  LIN {X -15849.996,Y 231.529,Z 80.709,A 172.46345,B 0.00000,C -180.00000} ; retreat
  ; Step 2908, bar 3026
  LIN {X -15449.996,Y 231.529,Z 999.647,A 172.46345,B 0.00000,C -180.00000} ; outside
  LIN {X -15449.996,Y 231.529,Z 30.709,A 172.46345,B 0.00000,C -180.00000} ; preinsert
  LIN {X -15449.996,Y 231.529,Z -219.291,A 172.46345,B 0.00000,C -180.00000} ; insert
  LIN {X -15449.996,Y 231.529,Z -219.291,A 172.46345,B 0.00000,C -180.00000} ; release
  LIN {X -15449.996,Y 231.529,Z 80.709,A 172.46345,B 0.00000,C -180.00000} ; retreat
  ; Step 2909, bar 3059
  LIN {X 15449.996,Y 231.529,Z 999.648,A 7.53655,B 0.00000,C 180.00000} ; outside
  LIN {X 15449.996,Y 231.529,Z 30.709,A 7.53655,B 0.00000,C 180.00000} ; preinsert
  LIN {X 15449.996,Y 231.529,Z -219.291,A 7.53655,B 0.00000,C 180.00000} ; insert
  LIN {X 15449.996,Y 231.529,Z -219.291,A 7.53655,B 0.00000,C 180.00000} ; release
  LIN {X 15449.996,Y 231.529,Z 80.709,A 7.53655,B 0.00000,C 180.00000} ; retreat
  ; Step 2910, bar 3065
  LIN {X 15849.996,Y 231.529,Z 999.648,A 7.53655,B 0.00000,C 180.00000} ; outside
  LIN {X 15849.996,Y 231.529,Z 30.709,A 7.53655,B 0.00000,C 180.00000} ; preinsert
  LIN {X 15849.996,Y 231.529,Z -219.291,A 7.53655,B 0.00000,C 180.00000} ; insert
  LIN {X 15849.996,Y 231.529,Z -219.291,A 7.53655,B 0.00000,C 180.00000} ; release
  LIN {X 15849.996,Y 231.529,Z 80.709,A 7.53655,B 0.00000,C 180.00000} ; retreat
  ; Step 2911, bar 3071
  LIN {X 16249.996,Y 231.529,Z 999.648,A 7.53655,B 0.00000,C 180.00000} ; outside
  LIN {X 16249.996,Y 231.529,Z 30.709,A 7.53655,B 0.00000,C 180.00000} ; preinsert
  LIN {X 16249.996,Y 231.529,Z -219.291,A 7.53655,B 0.00000,C 180.00000} ; insert
  LIN {X 16249.996,Y 231.529,Z -219.291,A 7.53655,B 0.00000,C 180.00000} ; release
  LIN {X 16249.996,Y 231.529,Z 80.709,A 7.53655,B 0.00000,C 180.00000} ; retreat
  ; Step 2912, bar 2635
  LIN {X -11999.916,Y -18.207,Z 1090.744,A -87.44234,B 0.00000,C 180.00000} ; outside
  LIN {X -11999.916,Y -18.207,Z 121.634,A -87.44234,B 0.00000,C 180.00000} ; preinsert
  LIN {X -11999.916,Y -18.207,Z -128.366,A -87.44234,B 0.00000,C 180.00000} ; insert
  LIN {X -11999.916,Y -18.207,Z -128.366,A -87.44234,B 0.00000,C 180.00000} ; release
  LIN {X -11999.916,Y -18.207,Z 171.634,A -87.44234,B 0.00000,C 180.00000} ; retreat
  ; Step 2913, bar 2629
  LIN {X -11249.916,Y -18.207,Z 1090.744,A -87.44234,B 0.00000,C 180.00000} ; outside
  LIN {X -11249.916,Y -18.207,Z 121.634,A -87.44234,B 0.00000,C 180.00000} ; preinsert
  LIN {X -11249.916,Y -18.207,Z -128.366,A -87.44234,B 0.00000,C 180.00000} ; insert
  LIN {X -11249.916,Y -18.207,Z -128.366,A -87.44234,B 0.00000,C 180.00000} ; release
  LIN {X -11249.916,Y -18.207,Z 171.634,A -87.44234,B 0.00000,C 180.00000} ; retreat
  ; Step 2914, bar 2622
  LIN {X -10499.916,Y -18.207,Z 1090.744,A -87.44234,B 0.00000,C 180.00000} ; outside
  LIN {X -10499.916,Y -18.207,Z 121.634,A -87.44234,B 0.00000,C 180.00000} ; preinsert
  LIN {X -10499.916,Y -18.207,Z -128.366,A -87.44234,B 0.00000,C 180.00000} ; insert
  LIN {X -10499.916,Y -18.207,Z -128.366,A -87.44234,B 0.00000,C 180.00000} ; release
  LIN {X -10499.916,Y -18.207,Z 171.634,A -87.44234,B 0.00000,C 180.00000} ; retreat
  ; Step 2915, bar 2615
  LIN {X -9749.916,Y -18.207,Z 1090.744,A -87.44234,B 0.00000,C 180.00000} ; outside
  LIN {X -9749.916,Y -18.207,Z 121.634,A -87.44234,B 0.00000,C 180.00000} ; preinsert
  LIN {X -9749.916,Y -18.207,Z -128.366,A -87.44234,B 0.00000,C 180.00000} ; insert
  LIN {X -9749.916,Y -18.207,Z -128.366,A -87.44234,B 0.00000,C 180.00000} ; release
  LIN {X -9749.916,Y -18.207,Z 171.634,A -87.44234,B 0.00000,C 180.00000} ; retreat
  ; Step 2916, bar 2608
  LIN {X -8999.916,Y -18.207,Z 1090.744,A -87.44234,B 0.00000,C 180.00000} ; outside
  LIN {X -8999.916,Y -18.207,Z 121.634,A -87.44234,B 0.00000,C 180.00000} ; preinsert
  LIN {X -8999.916,Y -18.207,Z -128.366,A -87.44234,B 0.00000,C 180.00000} ; insert
  LIN {X -8999.916,Y -18.207,Z -128.366,A -87.44234,B 0.00000,C 180.00000} ; release
  LIN {X -8999.916,Y -18.207,Z 171.634,A -87.44234,B 0.00000,C 180.00000} ; retreat
  ; Step 2917, bar 2601
  LIN {X -8249.916,Y -18.207,Z 1090.744,A -87.44234,B 0.00000,C 180.00000} ; outside
  LIN {X -8249.916,Y -18.207,Z 121.634,A -87.44234,B 0.00000,C 180.00000} ; preinsert
  LIN {X -8249.916,Y -18.207,Z -128.366,A -87.44234,B 0.00000,C 180.00000} ; insert
  LIN {X -8249.916,Y -18.207,Z -128.366,A -87.44234,B 0.00000,C 180.00000} ; release
  LIN {X -8249.916,Y -18.207,Z 171.634,A -87.44234,B 0.00000,C 180.00000} ; retreat
  ; Step 2918, bar 2594
  LIN {X -7499.916,Y -18.207,Z 1090.744,A -87.44234,B 0.00000,C 180.00000} ; outside
  LIN {X -7499.916,Y -18.207,Z 121.634,A -87.44234,B 0.00000,C 180.00000} ; preinsert
  LIN {X -7499.916,Y -18.207,Z -128.366,A -87.44234,B 0.00000,C 180.00000} ; insert
  LIN {X -7499.916,Y -18.207,Z -128.366,A -87.44234,B 0.00000,C 180.00000} ; release
  LIN {X -7499.916,Y -18.207,Z 171.634,A -87.44234,B 0.00000,C 180.00000} ; retreat
  ; Step 2919, bar 2587
  LIN {X -6749.916,Y -18.207,Z 1090.744,A -87.44234,B 0.00000,C 180.00000} ; outside
  LIN {X -6749.916,Y -18.207,Z 121.634,A -87.44234,B 0.00000,C 180.00000} ; preinsert
  LIN {X -6749.916,Y -18.207,Z -128.366,A -87.44234,B 0.00000,C 180.00000} ; insert
  LIN {X -6749.916,Y -18.207,Z -128.366,A -87.44234,B 0.00000,C 180.00000} ; release
  LIN {X -6749.916,Y -18.207,Z 171.634,A -87.44234,B 0.00000,C 180.00000} ; retreat
  ; Step 2920, bar 2580
  LIN {X -5999.916,Y -18.207,Z 1090.744,A -87.44234,B 0.00000,C 180.00000} ; outside
  LIN {X -5999.916,Y -18.207,Z 121.634,A -87.44234,B 0.00000,C 180.00000} ; preinsert
  LIN {X -5999.916,Y -18.207,Z -128.366,A -87.44234,B 0.00000,C 180.00000} ; insert
  LIN {X -5999.916,Y -18.207,Z -128.366,A -87.44234,B 0.00000,C 180.00000} ; release
  LIN {X -5999.916,Y -18.207,Z 171.634,A -87.44234,B 0.00000,C 180.00000} ; retreat
  ; Step 2921, bar 2573
  LIN {X -5249.916,Y -18.207,Z 1090.744,A -87.44234,B 0.00000,C 180.00000} ; outside
  LIN {X -5249.916,Y -18.207,Z 121.634,A -87.44234,B 0.00000,C 180.00000} ; preinsert
  LIN {X -5249.916,Y -18.207,Z -128.366,A -87.44234,B 0.00000,C 180.00000} ; insert
  LIN {X -5249.916,Y -18.207,Z -128.366,A -87.44234,B 0.00000,C 180.00000} ; release
  LIN {X -5249.916,Y -18.207,Z 171.634,A -87.44234,B 0.00000,C 180.00000} ; retreat
  ; Step 2922, bar 2566
  LIN {X -4499.916,Y -18.207,Z 1090.744,A -87.44234,B 0.00000,C 180.00000} ; outside
  LIN {X -4499.916,Y -18.207,Z 121.634,A -87.44234,B 0.00000,C 180.00000} ; preinsert
  LIN {X -4499.916,Y -18.207,Z -128.366,A -87.44234,B 0.00000,C 180.00000} ; insert
  LIN {X -4499.916,Y -18.207,Z -128.366,A -87.44234,B 0.00000,C 180.00000} ; release
  LIN {X -4499.916,Y -18.207,Z 171.634,A -87.44234,B 0.00000,C 180.00000} ; retreat
  ; Step 2923, bar 2559
  LIN {X -3749.916,Y -18.207,Z 1090.744,A -87.44234,B 0.00000,C 180.00000} ; outside
  LIN {X -3749.916,Y -18.207,Z 121.634,A -87.44234,B 0.00000,C 180.00000} ; preinsert
  LIN {X -3749.916,Y -18.207,Z -128.366,A -87.44234,B 0.00000,C 180.00000} ; insert
  LIN {X -3749.916,Y -18.207,Z -128.366,A -87.44234,B 0.00000,C 180.00000} ; release
  LIN {X -3749.916,Y -18.207,Z 171.634,A -87.44234,B 0.00000,C 180.00000} ; retreat
  ; Step 2924, bar 2552
  LIN {X -2999.916,Y -18.207,Z 1090.744,A -87.44234,B 0.00000,C 180.00000} ; outside
  LIN {X -2999.916,Y -18.207,Z 121.634,A -87.44234,B 0.00000,C 180.00000} ; preinsert
  LIN {X -2999.916,Y -18.207,Z -128.366,A -87.44234,B 0.00000,C 180.00000} ; insert
  LIN {X -2999.916,Y -18.207,Z -128.366,A -87.44234,B 0.00000,C 180.00000} ; release
  LIN {X -2999.916,Y -18.207,Z 171.634,A -87.44234,B 0.00000,C 180.00000} ; retreat
  ; Step 2925, bar 2545
  LIN {X -2249.916,Y -18.207,Z 1090.744,A -87.44234,B 0.00000,C 180.00000} ; outside
  LIN {X -2249.916,Y -18.207,Z 121.634,A -87.44234,B 0.00000,C 180.00000} ; preinsert
  LIN {X -2249.916,Y -18.207,Z -128.366,A -87.44234,B 0.00000,C 180.00000} ; insert
  LIN {X -2249.916,Y -18.207,Z -128.366,A -87.44234,B 0.00000,C 180.00000} ; release
  LIN {X -2249.916,Y -18.207,Z 171.634,A -87.44234,B 0.00000,C 180.00000} ; retreat
  ; Step 2926, bar 2538
  LIN {X -1499.916,Y -18.207,Z 1090.744,A -87.44234,B 0.00000,C 180.00000} ; outside
  LIN {X -1499.916,Y -18.207,Z 121.634,A -87.44234,B 0.00000,C 180.00000} ; preinsert
  LIN {X -1499.916,Y -18.207,Z -128.366,A -87.44234,B 0.00000,C 180.00000} ; insert
  LIN {X -1499.916,Y -18.207,Z -128.366,A -87.44234,B 0.00000,C 180.00000} ; release
  LIN {X -1499.916,Y -18.207,Z 171.634,A -87.44234,B 0.00000,C 180.00000} ; retreat
  ; Step 2927, bar 1972
  LIN {X 0.084,Y -18.207,Z 1090.744,A -87.44234,B 0.00000,C -180.00000} ; outside
  LIN {X 0.084,Y -18.207,Z 121.634,A -87.44234,B 0.00000,C -180.00000} ; preinsert
  LIN {X 0.084,Y -18.207,Z -128.366,A -87.44234,B 0.00000,C -180.00000} ; insert
  LIN {X 0.084,Y -18.207,Z -128.366,A -87.44234,B 0.00000,C -180.00000} ; release
  LIN {X 0.084,Y -18.207,Z 171.634,A -87.44234,B 0.00000,C -180.00000} ; retreat
  ; Step 2928, bar 2691
  LIN {X 1499.916,Y -18.207,Z 1090.744,A -92.55766,B 0.00000,C -180.00000} ; outside
  LIN {X 1499.916,Y -18.207,Z 121.634,A -92.55766,B 0.00000,C -180.00000} ; preinsert
  LIN {X 1499.916,Y -18.207,Z -128.366,A -92.55766,B 0.00000,C -180.00000} ; insert
  LIN {X 1499.916,Y -18.207,Z -128.366,A -92.55766,B 0.00000,C -180.00000} ; release
  LIN {X 1499.916,Y -18.207,Z 171.634,A -92.55766,B 0.00000,C -180.00000} ; retreat
  ; Step 2929, bar 2695
  LIN {X 2249.916,Y -18.207,Z 1090.744,A -92.55766,B 0.00000,C -180.00000} ; outside
  LIN {X 2249.916,Y -18.207,Z 121.634,A -92.55766,B 0.00000,C -180.00000} ; preinsert
  LIN {X 2249.916,Y -18.207,Z -128.366,A -92.55766,B 0.00000,C -180.00000} ; insert
  LIN {X 2249.916,Y -18.207,Z -128.366,A -92.55766,B 0.00000,C -180.00000} ; release
  LIN {X 2249.916,Y -18.207,Z 171.634,A -92.55766,B 0.00000,C -180.00000} ; retreat
  ; Step 2930, bar 2699
  LIN {X 2999.916,Y -18.207,Z 1090.744,A -92.55766,B 0.00000,C -180.00000} ; outside
  LIN {X 2999.916,Y -18.207,Z 121.634,A -92.55766,B 0.00000,C -180.00000} ; preinsert
  LIN {X 2999.916,Y -18.207,Z -128.366,A -92.55766,B 0.00000,C -180.00000} ; insert
  LIN {X 2999.916,Y -18.207,Z -128.366,A -92.55766,B 0.00000,C -180.00000} ; release
  LIN {X 2999.916,Y -18.207,Z 171.634,A -92.55766,B 0.00000,C -180.00000} ; retreat
  ; Step 2931, bar 2703
  LIN {X 3749.916,Y -18.207,Z 1090.744,A -92.55766,B 0.00000,C -180.00000} ; outside
  LIN {X 3749.916,Y -18.207,Z 121.634,A -92.55766,B 0.00000,C -180.00000} ; preinsert
  LIN {X 3749.916,Y -18.207,Z -128.366,A -92.55766,B 0.00000,C -180.00000} ; insert
  LIN {X 3749.916,Y -18.207,Z -128.366,A -92.55766,B 0.00000,C -180.00000} ; release
  LIN {X 3749.916,Y -18.207,Z 171.634,A -92.55766,B 0.00000,C -180.00000} ; retreat
  ; Step 2932, bar 2707
  LIN {X 4499.916,Y -18.207,Z 1090.744,A -92.55766,B 0.00000,C -180.00000} ; outside
  LIN {X 4499.916,Y -18.207,Z 121.634,A -92.55766,B 0.00000,C -180.00000} ; preinsert
  LIN {X 4499.916,Y -18.207,Z -128.366,A -92.55766,B 0.00000,C -180.00000} ; insert
  LIN {X 4499.916,Y -18.207,Z -128.366,A -92.55766,B 0.00000,C -180.00000} ; release
  LIN {X 4499.916,Y -18.207,Z 171.634,A -92.55766,B 0.00000,C -180.00000} ; retreat
  ; Step 2933, bar 2711
  LIN {X 5249.916,Y -18.207,Z 1090.744,A -92.55766,B 0.00000,C -180.00000} ; outside
  LIN {X 5249.916,Y -18.207,Z 121.634,A -92.55766,B 0.00000,C -180.00000} ; preinsert
  LIN {X 5249.916,Y -18.207,Z -128.366,A -92.55766,B 0.00000,C -180.00000} ; insert
  LIN {X 5249.916,Y -18.207,Z -128.366,A -92.55766,B 0.00000,C -180.00000} ; release
  LIN {X 5249.916,Y -18.207,Z 171.634,A -92.55766,B 0.00000,C -180.00000} ; retreat
  ; Step 2934, bar 2715
  LIN {X 5999.916,Y -18.207,Z 1090.744,A -92.55766,B 0.00000,C -180.00000} ; outside
  LIN {X 5999.916,Y -18.207,Z 121.634,A -92.55766,B 0.00000,C -180.00000} ; preinsert
  LIN {X 5999.916,Y -18.207,Z -128.366,A -92.55766,B 0.00000,C -180.00000} ; insert
  LIN {X 5999.916,Y -18.207,Z -128.366,A -92.55766,B 0.00000,C -180.00000} ; release
  LIN {X 5999.916,Y -18.207,Z 171.634,A -92.55766,B 0.00000,C -180.00000} ; retreat
  ; Step 2935, bar 2719
  LIN {X 6749.916,Y -18.207,Z 1090.744,A -92.55766,B 0.00000,C -180.00000} ; outside
  LIN {X 6749.916,Y -18.207,Z 121.634,A -92.55766,B 0.00000,C -180.00000} ; preinsert
  LIN {X 6749.916,Y -18.207,Z -128.366,A -92.55766,B 0.00000,C -180.00000} ; insert
  LIN {X 6749.916,Y -18.207,Z -128.366,A -92.55766,B 0.00000,C -180.00000} ; release
  LIN {X 6749.916,Y -18.207,Z 171.634,A -92.55766,B 0.00000,C -180.00000} ; retreat
  ; Step 2936, bar 2723
  LIN {X 7499.916,Y -18.207,Z 1090.744,A -92.55766,B 0.00000,C -180.00000} ; outside
  LIN {X 7499.916,Y -18.207,Z 121.634,A -92.55766,B 0.00000,C -180.00000} ; preinsert
  LIN {X 7499.916,Y -18.207,Z -128.366,A -92.55766,B 0.00000,C -180.00000} ; insert
  LIN {X 7499.916,Y -18.207,Z -128.366,A -92.55766,B 0.00000,C -180.00000} ; release
  LIN {X 7499.916,Y -18.207,Z 171.634,A -92.55766,B 0.00000,C -180.00000} ; retreat
  ; Step 2937, bar 2727
  LIN {X 8249.916,Y -18.207,Z 1090.744,A -92.55766,B 0.00000,C -180.00000} ; outside
  LIN {X 8249.916,Y -18.207,Z 121.634,A -92.55766,B 0.00000,C -180.00000} ; preinsert
  LIN {X 8249.916,Y -18.207,Z -128.366,A -92.55766,B 0.00000,C -180.00000} ; insert
  LIN {X 8249.916,Y -18.207,Z -128.366,A -92.55766,B 0.00000,C -180.00000} ; release
  LIN {X 8249.916,Y -18.207,Z 171.634,A -92.55766,B 0.00000,C -180.00000} ; retreat
  ; Step 2938, bar 2731
  LIN {X 8999.916,Y -18.207,Z 1090.744,A -92.55766,B 0.00000,C -180.00000} ; outside
  LIN {X 8999.916,Y -18.207,Z 121.634,A -92.55766,B 0.00000,C -180.00000} ; preinsert
  LIN {X 8999.916,Y -18.207,Z -128.366,A -92.55766,B 0.00000,C -180.00000} ; insert
  LIN {X 8999.916,Y -18.207,Z -128.366,A -92.55766,B 0.00000,C -180.00000} ; release
  LIN {X 8999.916,Y -18.207,Z 171.634,A -92.55766,B 0.00000,C -180.00000} ; retreat
  ; Step 2939, bar 2735
  LIN {X 9749.916,Y -18.207,Z 1090.744,A -92.55766,B 0.00000,C -180.00000} ; outside
  LIN {X 9749.916,Y -18.207,Z 121.634,A -92.55766,B 0.00000,C -180.00000} ; preinsert
  LIN {X 9749.916,Y -18.207,Z -128.366,A -92.55766,B 0.00000,C -180.00000} ; insert
  LIN {X 9749.916,Y -18.207,Z -128.366,A -92.55766,B 0.00000,C -180.00000} ; release
  LIN {X 9749.916,Y -18.207,Z 171.634,A -92.55766,B 0.00000,C -180.00000} ; retreat
  ; Step 2940, bar 2739
  LIN {X 10499.916,Y -18.207,Z 1090.744,A -92.55766,B 0.00000,C -180.00000} ; outside
  LIN {X 10499.916,Y -18.207,Z 121.634,A -92.55766,B 0.00000,C -180.00000} ; preinsert
  LIN {X 10499.916,Y -18.207,Z -128.366,A -92.55766,B 0.00000,C -180.00000} ; insert
  LIN {X 10499.916,Y -18.207,Z -128.366,A -92.55766,B 0.00000,C -180.00000} ; release
  LIN {X 10499.916,Y -18.207,Z 171.634,A -92.55766,B 0.00000,C -180.00000} ; retreat
  ; Step 2941, bar 2743
  LIN {X 11249.916,Y -18.207,Z 1090.744,A -92.55766,B 0.00000,C -180.00000} ; outside
  LIN {X 11249.916,Y -18.207,Z 121.634,A -92.55766,B 0.00000,C -180.00000} ; preinsert
  LIN {X 11249.916,Y -18.207,Z -128.366,A -92.55766,B 0.00000,C -180.00000} ; insert
  LIN {X 11249.916,Y -18.207,Z -128.366,A -92.55766,B 0.00000,C -180.00000} ; release
  LIN {X 11249.916,Y -18.207,Z 171.634,A -92.55766,B 0.00000,C -180.00000} ; retreat
  ; Step 2942, bar 2747
  LIN {X 11999.916,Y -18.207,Z 1090.744,A -92.55766,B 0.00000,C -180.00000} ; outside
  LIN {X 11999.916,Y -18.207,Z 121.634,A -92.55766,B 0.00000,C -180.00000} ; preinsert
  LIN {X 11999.916,Y -18.207,Z -128.366,A -92.55766,B 0.00000,C -180.00000} ; insert
  LIN {X 11999.916,Y -18.207,Z -128.366,A -92.55766,B 0.00000,C -180.00000} ; release
  LIN {X 11999.916,Y -18.207,Z 171.634,A -92.55766,B 0.00000,C -180.00000} ; retreat
  ; Step 2943, bar 2687
  LIN {X 749.916,Y -18.207,Z 1090.744,A -92.55766,B 0.00000,C -180.00000} ; outside
  LIN {X 749.916,Y -18.207,Z 121.634,A -92.55766,B 0.00000,C -180.00000} ; preinsert
  LIN {X 749.916,Y -18.207,Z -128.366,A -92.55766,B 0.00000,C -180.00000} ; insert
  LIN {X 749.916,Y -18.207,Z -128.366,A -92.55766,B 0.00000,C -180.00000} ; release
  LIN {X 749.916,Y -18.207,Z 171.634,A -92.55766,B 0.00000,C -180.00000} ; retreat
  ; Step 2944, bar 2531
  LIN {X -749.916,Y -18.207,Z 1090.744,A -87.44234,B 0.00000,C 180.00000} ; outside
  LIN {X -749.916,Y -18.207,Z 121.634,A -87.44234,B 0.00000,C 180.00000} ; preinsert
  LIN {X -749.916,Y -18.207,Z -128.366,A -87.44234,B 0.00000,C 180.00000} ; insert
  LIN {X -749.916,Y -18.207,Z -128.366,A -87.44234,B 0.00000,C 180.00000} ; release
  LIN {X -749.916,Y -18.207,Z 171.634,A -87.44234,B 0.00000,C 180.00000} ; retreat
  ; Step 2945, bar 3056
  LIN {X 15249.996,Y -18.471,Z 1010.647,A 7.53655,B 0.00000,C 180.00000} ; outside
  LIN {X 15249.996,Y -18.471,Z 36.610,A 7.53655,B 0.00000,C 180.00000} ; preinsert
  LIN {X 15249.996,Y -18.471,Z -213.390,A 7.53655,B 0.00000,C 180.00000} ; insert
  LIN {X 15249.996,Y -18.471,Z -213.390,A 7.53655,B 0.00000,C 180.00000} ; release
  LIN {X 15249.996,Y -18.471,Z 86.610,A 7.53655,B 0.00000,C 180.00000} ; retreat
  ; Step 2946, bar 3062
  LIN {X 15649.996,Y -18.471,Z 1010.647,A 7.53655,B 0.00000,C 180.00000} ; outside
  LIN {X 15649.996,Y -18.471,Z 36.610,A 7.53655,B 0.00000,C 180.00000} ; preinsert
  LIN {X 15649.996,Y -18.471,Z -213.390,A 7.53655,B 0.00000,C 180.00000} ; insert
  LIN {X 15649.996,Y -18.471,Z -213.390,A 7.53655,B 0.00000,C 180.00000} ; release
  LIN {X 15649.996,Y -18.471,Z 86.610,A 7.53655,B 0.00000,C 180.00000} ; retreat
  ; Step 2947, bar 3068
  LIN {X 16049.996,Y -18.471,Z 1010.647,A 7.53655,B 0.00000,C 180.00000} ; outside
  LIN {X 16049.996,Y -18.471,Z 36.610,A 7.53655,B 0.00000,C 180.00000} ; preinsert
  LIN {X 16049.996,Y -18.471,Z -213.390,A 7.53655,B 0.00000,C 180.00000} ; insert
  LIN {X 16049.996,Y -18.471,Z -213.390,A 7.53655,B 0.00000,C 180.00000} ; release
  LIN {X 16049.996,Y -18.471,Z 86.610,A 7.53655,B 0.00000,C 180.00000} ; retreat
  ; Step 2948, bar 3035
  LIN {X -16049.996,Y -18.471,Z 1010.647,A 172.46345,B 0.00000,C 180.00000} ; outside
  LIN {X -16049.996,Y -18.471,Z 36.610,A 172.46345,B 0.00000,C 180.00000} ; preinsert
  LIN {X -16049.996,Y -18.471,Z -213.390,A 172.46345,B 0.00000,C 180.00000} ; insert
  LIN {X -16049.996,Y -18.471,Z -213.390,A 172.46345,B 0.00000,C 180.00000} ; release
  LIN {X -16049.996,Y -18.471,Z 86.610,A 172.46345,B 0.00000,C 180.00000} ; retreat
  ; Step 2949, bar 3029
  LIN {X -15649.996,Y -18.471,Z 1010.647,A 172.46345,B 0.00000,C 180.00000} ; outside
  LIN {X -15649.996,Y -18.471,Z 36.610,A 172.46345,B 0.00000,C 180.00000} ; preinsert
  LIN {X -15649.996,Y -18.471,Z -213.390,A 172.46345,B 0.00000,C 180.00000} ; insert
  LIN {X -15649.996,Y -18.471,Z -213.390,A 172.46345,B 0.00000,C 180.00000} ; release
  LIN {X -15649.996,Y -18.471,Z 86.610,A 172.46345,B 0.00000,C 180.00000} ; retreat
  ; Step 2950, bar 3023
  LIN {X -15249.996,Y -18.471,Z 1010.647,A 172.46345,B 0.00000,C 180.00000} ; outside
  LIN {X -15249.996,Y -18.471,Z 36.610,A 172.46345,B 0.00000,C 180.00000} ; preinsert
  LIN {X -15249.996,Y -18.471,Z -213.390,A 172.46345,B 0.00000,C 180.00000} ; insert
  LIN {X -15249.996,Y -18.471,Z -213.390,A 172.46345,B 0.00000,C 180.00000} ; release
  LIN {X -15249.996,Y -18.471,Z 86.610,A 172.46345,B 0.00000,C 180.00000} ; retreat
  ; Step 2951, bar 1530
  LIN {X 1986.216,Y 1384.682,Z 869.354,A -90.02766,B 0.00000,C -180.00000} ; outside
  LIN {X 1986.216,Y 1384.682,Z -118.655,A -90.02766,B 0.00000,C -180.00000} ; preinsert
  LIN {X 1986.216,Y 1384.682,Z -368.655,A -90.02766,B 0.00000,C -180.00000} ; insert
  LIN {X 1986.216,Y 1384.682,Z -368.655,A -90.02766,B 0.00000,C -180.00000} ; release
  LIN {X 1986.216,Y 1384.682,Z -68.655,A -90.02766,B 0.00000,C -180.00000} ; retreat
  ; Step 2952, bar 1532
  LIN {X 5986.216,Y 1384.682,Z 869.354,A -90.02766,B 0.00000,C 180.00000} ; outside
  LIN {X 5986.216,Y 1384.682,Z -118.655,A -90.02766,B 0.00000,C 180.00000} ; preinsert
  LIN {X 5986.216,Y 1384.682,Z -368.655,A -90.02766,B 0.00000,C 180.00000} ; insert
  LIN {X 5986.216,Y 1384.682,Z -368.655,A -90.02766,B 0.00000,C 180.00000} ; release
  LIN {X 5986.216,Y 1384.682,Z -68.655,A -90.02766,B 0.00000,C 180.00000} ; retreat
  ; Step 2953, bar 1534
  LIN {X 9986.216,Y 1384.682,Z 869.354,A -90.02766,B 0.00000,C -180.00000} ; outside
  LIN {X 9986.216,Y 1384.682,Z -118.655,A -90.02766,B 0.00000,C -180.00000} ; preinsert
  LIN {X 9986.216,Y 1384.682,Z -368.655,A -90.02766,B 0.00000,C -180.00000} ; insert
  LIN {X 9986.216,Y 1384.682,Z -368.655,A -90.02766,B 0.00000,C -180.00000} ; release
  LIN {X 9986.216,Y 1384.682,Z -68.655,A -90.02766,B 0.00000,C -180.00000} ; retreat
  ; Step 2954, bar 1536
  LIN {X 13936.216,Y 1384.682,Z 869.354,A -90.02766,B 0.00000,C -180.00000} ; outside
  LIN {X 13936.216,Y 1384.682,Z -118.655,A -90.02766,B 0.00000,C -180.00000} ; preinsert
  LIN {X 13936.216,Y 1384.682,Z -368.655,A -90.02766,B 0.00000,C -180.00000} ; insert
  LIN {X 13936.216,Y 1384.682,Z -368.655,A -90.02766,B 0.00000,C -180.00000} ; release
  LIN {X 13936.216,Y 1384.682,Z -68.655,A -90.02766,B 0.00000,C -180.00000} ; retreat
  ; Step 2955, bar 1538
  LIN {X 14036.216,Y 1384.682,Z 869.354,A -90.02766,B 0.00000,C -180.00000} ; outside
  LIN {X 14036.216,Y 1384.682,Z -118.655,A -90.02766,B 0.00000,C -180.00000} ; preinsert
  LIN {X 14036.216,Y 1384.682,Z -368.655,A -90.02766,B 0.00000,C -180.00000} ; insert
  LIN {X 14036.216,Y 1384.682,Z -368.655,A -90.02766,B 0.00000,C -180.00000} ; release
  LIN {X 14036.216,Y 1384.682,Z -68.655,A -90.02766,B 0.00000,C -180.00000} ; retreat
  ; Step 2956, bar 1549
  LIN {X -1986.216,Y -1384.682,Z 869.354,A 89.97234,B 0.00000,C 180.00000} ; outside
  LIN {X -1986.216,Y -1384.682,Z -118.655,A 89.97234,B 0.00000,C 180.00000} ; preinsert
  LIN {X -1986.216,Y -1384.682,Z -368.655,A 89.97234,B 0.00000,C 180.00000} ; insert
  LIN {X -1986.216,Y -1384.682,Z -368.655,A 89.97234,B 0.00000,C 180.00000} ; release
  LIN {X -1986.216,Y -1384.682,Z -68.655,A 89.97234,B 0.00000,C 180.00000} ; retreat
  ; Step 2957, bar 1551
  LIN {X -5986.216,Y -1384.682,Z 869.354,A 89.97234,B 0.00000,C 180.00000} ; outside
  LIN {X -5986.216,Y -1384.682,Z -118.655,A 89.97234,B 0.00000,C 180.00000} ; preinsert
  LIN {X -5986.216,Y -1384.682,Z -368.655,A 89.97234,B 0.00000,C 180.00000} ; insert
  LIN {X -5986.216,Y -1384.682,Z -368.655,A 89.97234,B 0.00000,C 180.00000} ; release
  LIN {X -5986.216,Y -1384.682,Z -68.655,A 89.97234,B 0.00000,C 180.00000} ; retreat
  ; Step 2958, bar 1553
  LIN {X -9986.216,Y -1384.682,Z 869.354,A 89.97234,B 0.00000,C -180.00000} ; outside
  LIN {X -9986.216,Y -1384.682,Z -118.655,A 89.97234,B 0.00000,C -180.00000} ; preinsert
  LIN {X -9986.216,Y -1384.682,Z -368.655,A 89.97234,B 0.00000,C -180.00000} ; insert
  LIN {X -9986.216,Y -1384.682,Z -368.655,A 89.97234,B 0.00000,C -180.00000} ; release
  LIN {X -9986.216,Y -1384.682,Z -68.655,A 89.97234,B 0.00000,C -180.00000} ; retreat
  ; Step 2959, bar 1555
  LIN {X -13936.216,Y -1384.682,Z 869.354,A 89.97234,B 0.00000,C -180.00000} ; outside
  LIN {X -13936.216,Y -1384.682,Z -118.655,A 89.97234,B 0.00000,C -180.00000} ; preinsert
  LIN {X -13936.216,Y -1384.682,Z -368.655,A 89.97234,B 0.00000,C -180.00000} ; insert
  LIN {X -13936.216,Y -1384.682,Z -368.655,A 89.97234,B 0.00000,C -180.00000} ; release
  LIN {X -13936.216,Y -1384.682,Z -68.655,A 89.97234,B 0.00000,C -180.00000} ; retreat
  ; Step 2960, bar 1557
  LIN {X -14036.216,Y -1384.682,Z 869.354,A 89.97234,B 0.00000,C -180.00000} ; outside
  LIN {X -14036.216,Y -1384.682,Z -118.655,A 89.97234,B 0.00000,C -180.00000} ; preinsert
  LIN {X -14036.216,Y -1384.682,Z -368.655,A 89.97234,B 0.00000,C -180.00000} ; insert
  LIN {X -14036.216,Y -1384.682,Z -368.655,A 89.97234,B 0.00000,C -180.00000} ; release
  LIN {X -14036.216,Y -1384.682,Z -68.655,A 89.97234,B 0.00000,C -180.00000} ; retreat
  ; Step 2961, bar 1529
  LIN {X 1986.216,Y -1384.663,Z 869.359,A 90.02766,B 0.00000,C 180.00000} ; outside
  LIN {X 1986.216,Y -1384.663,Z -118.650,A 90.02766,B 0.00000,C 180.00000} ; preinsert
  LIN {X 1986.216,Y -1384.663,Z -368.650,A 90.02766,B 0.00000,C 180.00000} ; insert
  LIN {X 1986.216,Y -1384.663,Z -368.650,A 90.02766,B 0.00000,C 180.00000} ; release
  LIN {X 1986.216,Y -1384.663,Z -68.650,A 90.02766,B 0.00000,C 180.00000} ; retreat
  ; Step 2962, bar 1531
  LIN {X 5986.216,Y -1384.663,Z 869.359,A 90.02766,B 0.00000,C 180.00000} ; outside
  LIN {X 5986.216,Y -1384.663,Z -118.650,A 90.02766,B 0.00000,C 180.00000} ; preinsert
  LIN {X 5986.216,Y -1384.663,Z -368.650,A 90.02766,B 0.00000,C 180.00000} ; insert
  LIN {X 5986.216,Y -1384.663,Z -368.650,A 90.02766,B 0.00000,C 180.00000} ; release
  LIN {X 5986.216,Y -1384.663,Z -68.650,A 90.02766,B 0.00000,C 180.00000} ; retreat
  ; Step 2963, bar 1533
  LIN {X 9986.216,Y -1384.663,Z 869.359,A 90.02766,B 0.00000,C -180.00000} ; outside
  LIN {X 9986.216,Y -1384.663,Z -118.650,A 90.02766,B 0.00000,C -180.00000} ; preinsert
  LIN {X 9986.216,Y -1384.663,Z -368.650,A 90.02766,B 0.00000,C -180.00000} ; insert
  LIN {X 9986.216,Y -1384.663,Z -368.650,A 90.02766,B 0.00000,C -180.00000} ; release
  LIN {X 9986.216,Y -1384.663,Z -68.650,A 90.02766,B 0.00000,C -180.00000} ; retreat
  ; Step 2964, bar 1535
  LIN {X 13936.216,Y -1384.663,Z 869.359,A 90.02766,B 0.00000,C -180.00000} ; outside
  LIN {X 13936.216,Y -1384.663,Z -118.650,A 90.02766,B 0.00000,C -180.00000} ; preinsert
  LIN {X 13936.216,Y -1384.663,Z -368.650,A 90.02766,B 0.00000,C -180.00000} ; insert
  LIN {X 13936.216,Y -1384.663,Z -368.650,A 90.02766,B 0.00000,C -180.00000} ; release
  LIN {X 13936.216,Y -1384.663,Z -68.650,A 90.02766,B 0.00000,C -180.00000} ; retreat
  ; Step 2965, bar 1537
  LIN {X 14036.216,Y -1384.663,Z 869.359,A 90.02766,B 0.00000,C -180.00000} ; outside
  LIN {X 14036.216,Y -1384.663,Z -118.650,A 90.02766,B 0.00000,C -180.00000} ; preinsert
  LIN {X 14036.216,Y -1384.663,Z -368.650,A 90.02766,B 0.00000,C -180.00000} ; insert
  LIN {X 14036.216,Y -1384.663,Z -368.650,A 90.02766,B 0.00000,C -180.00000} ; release
  LIN {X 14036.216,Y -1384.663,Z -68.650,A 90.02766,B 0.00000,C -180.00000} ; retreat
  ; Step 2966, bar 1550
  LIN {X -1986.216,Y 1384.663,Z 869.359,A -89.97234,B 0.00000,C 180.00000} ; outside
  LIN {X -1986.216,Y 1384.663,Z -118.650,A -89.97234,B 0.00000,C 180.00000} ; preinsert
  LIN {X -1986.216,Y 1384.663,Z -368.650,A -89.97234,B 0.00000,C 180.00000} ; insert
  LIN {X -1986.216,Y 1384.663,Z -368.650,A -89.97234,B 0.00000,C 180.00000} ; release
  LIN {X -1986.216,Y 1384.663,Z -68.650,A -89.97234,B 0.00000,C 180.00000} ; retreat
  ; Step 2967, bar 1552
  LIN {X -5986.216,Y 1384.663,Z 869.359,A -89.97234,B 0.00000,C 180.00000} ; outside
  LIN {X -5986.216,Y 1384.663,Z -118.650,A -89.97234,B 0.00000,C 180.00000} ; preinsert
  LIN {X -5986.216,Y 1384.663,Z -368.650,A -89.97234,B 0.00000,C 180.00000} ; insert
  LIN {X -5986.216,Y 1384.663,Z -368.650,A -89.97234,B 0.00000,C 180.00000} ; release
  LIN {X -5986.216,Y 1384.663,Z -68.650,A -89.97234,B 0.00000,C 180.00000} ; retreat
  ; Step 2968, bar 1554
  LIN {X -9986.216,Y 1384.663,Z 869.359,A -89.97234,B 0.00000,C 180.00000} ; outside
  LIN {X -9986.216,Y 1384.663,Z -118.650,A -89.97234,B 0.00000,C 180.00000} ; preinsert
  LIN {X -9986.216,Y 1384.663,Z -368.650,A -89.97234,B 0.00000,C 180.00000} ; insert
  LIN {X -9986.216,Y 1384.663,Z -368.650,A -89.97234,B 0.00000,C 180.00000} ; release
  LIN {X -9986.216,Y 1384.663,Z -68.650,A -89.97234,B 0.00000,C 180.00000} ; retreat
  ; Step 2969, bar 1556
  LIN {X -13936.216,Y 1384.663,Z 869.359,A -89.97234,B 0.00000,C 180.00000} ; outside
  LIN {X -13936.216,Y 1384.663,Z -118.650,A -89.97234,B 0.00000,C 180.00000} ; preinsert
  LIN {X -13936.216,Y 1384.663,Z -368.650,A -89.97234,B 0.00000,C 180.00000} ; insert
  LIN {X -13936.216,Y 1384.663,Z -368.650,A -89.97234,B 0.00000,C 180.00000} ; release
  LIN {X -13936.216,Y 1384.663,Z -68.650,A -89.97234,B 0.00000,C 180.00000} ; retreat
  ; Step 2970, bar 1558
  LIN {X -14036.216,Y 1384.663,Z 869.359,A -89.97234,B 0.00000,C 180.00000} ; outside
  LIN {X -14036.216,Y 1384.663,Z -118.650,A -89.97234,B 0.00000,C 180.00000} ; preinsert
  LIN {X -14036.216,Y 1384.663,Z -368.650,A -89.97234,B 0.00000,C 180.00000} ; insert
  LIN {X -14036.216,Y 1384.663,Z -368.650,A -89.97234,B 0.00000,C 180.00000} ; release
  LIN {X -14036.216,Y 1384.663,Z -68.650,A -89.97234,B 0.00000,C 180.00000} ; retreat
  ; Step 2971, bar 1251
  LIN {X -14.107,Y -2029.899,Z 855.478,A 89.96659,B 0.00000,C 180.00000} ; outside
  LIN {X -14.107,Y -2029.899,Z -132.531,A 89.96659,B 0.00000,C 180.00000} ; preinsert
  LIN {X -14.107,Y -2029.899,Z -382.531,A 89.96659,B 0.00000,C 180.00000} ; insert
  LIN {X -14.107,Y -2029.899,Z -382.531,A 89.96659,B 0.00000,C 180.00000} ; release
  LIN {X -14.107,Y -2029.899,Z -82.531,A 89.96659,B 0.00000,C 180.00000} ; retreat
  ; Step 2972, bar 1253
  LIN {X 110.893,Y -2029.899,Z 855.478,A 89.96659,B 0.00000,C 180.00000} ; outside
  LIN {X 110.893,Y -2029.899,Z -132.531,A 89.96659,B 0.00000,C 180.00000} ; preinsert
  LIN {X 110.893,Y -2029.899,Z -382.531,A 89.96659,B 0.00000,C 180.00000} ; insert
  LIN {X 110.893,Y -2029.899,Z -382.531,A 89.96659,B 0.00000,C 180.00000} ; release
  LIN {X 110.893,Y -2029.899,Z -82.531,A 89.96659,B 0.00000,C 180.00000} ; retreat
  ; Step 2973, bar 1255
  LIN {X 235.893,Y -2029.899,Z 855.478,A 89.96659,B 0.00000,C 180.00000} ; outside
  LIN {X 235.893,Y -2029.899,Z -132.531,A 89.96659,B 0.00000,C 180.00000} ; preinsert
  LIN {X 235.893,Y -2029.899,Z -382.531,A 89.96659,B 0.00000,C 180.00000} ; insert
  LIN {X 235.893,Y -2029.899,Z -382.531,A 89.96659,B 0.00000,C 180.00000} ; release
  LIN {X 235.893,Y -2029.899,Z -82.531,A 89.96659,B 0.00000,C 180.00000} ; retreat
  ; Step 2974, bar 1257
  LIN {X 360.893,Y -2029.899,Z 855.478,A 89.96659,B 0.00000,C 180.00000} ; outside
  LIN {X 360.893,Y -2029.899,Z -132.531,A 89.96659,B 0.00000,C 180.00000} ; preinsert
  LIN {X 360.893,Y -2029.899,Z -382.531,A 89.96659,B 0.00000,C 180.00000} ; insert
  LIN {X 360.893,Y -2029.899,Z -382.531,A 89.96659,B 0.00000,C 180.00000} ; release
  LIN {X 360.893,Y -2029.899,Z -82.531,A 89.96659,B 0.00000,C 180.00000} ; retreat
  ; Step 2975, bar 1259
  LIN {X 485.893,Y -2029.899,Z 855.478,A 89.96659,B 0.00000,C 180.00000} ; outside
  LIN {X 485.893,Y -2029.899,Z -132.531,A 89.96659,B 0.00000,C 180.00000} ; preinsert
  LIN {X 485.893,Y -2029.899,Z -382.531,A 89.96659,B 0.00000,C 180.00000} ; insert
  LIN {X 485.893,Y -2029.899,Z -382.531,A 89.96659,B 0.00000,C 180.00000} ; release
  LIN {X 485.893,Y -2029.899,Z -82.531,A 89.96659,B 0.00000,C 180.00000} ; retreat
  ; Step 2976, bar 1261
  LIN {X 610.893,Y -2029.899,Z 855.478,A 89.96659,B 0.00000,C 180.00000} ; outside
  LIN {X 610.893,Y -2029.899,Z -132.531,A 89.96659,B 0.00000,C 180.00000} ; preinsert
  LIN {X 610.893,Y -2029.899,Z -382.531,A 89.96659,B 0.00000,C 180.00000} ; insert
  LIN {X 610.893,Y -2029.899,Z -382.531,A 89.96659,B 0.00000,C 180.00000} ; release
  LIN {X 610.893,Y -2029.899,Z -82.531,A 89.96659,B 0.00000,C 180.00000} ; retreat
  ; Step 2977, bar 1263
  LIN {X 735.893,Y -2029.899,Z 855.478,A 89.96659,B 0.00000,C 180.00000} ; outside
  LIN {X 735.893,Y -2029.899,Z -132.531,A 89.96659,B 0.00000,C 180.00000} ; preinsert
  LIN {X 735.893,Y -2029.899,Z -382.531,A 89.96659,B 0.00000,C 180.00000} ; insert
  LIN {X 735.893,Y -2029.899,Z -382.531,A 89.96659,B 0.00000,C 180.00000} ; release
  LIN {X 735.893,Y -2029.899,Z -82.531,A 89.96659,B 0.00000,C 180.00000} ; retreat
  ; Step 2978, bar 1265
  LIN {X 860.893,Y -2029.899,Z 855.478,A 89.96659,B 0.00000,C 180.00000} ; outside
  LIN {X 860.893,Y -2029.899,Z -132.531,A 89.96659,B 0.00000,C 180.00000} ; preinsert
  LIN {X 860.893,Y -2029.899,Z -382.531,A 89.96659,B 0.00000,C 180.00000} ; insert
  LIN {X 860.893,Y -2029.899,Z -382.531,A 89.96659,B 0.00000,C 180.00000} ; release
  LIN {X 860.893,Y -2029.899,Z -82.531,A 89.96659,B 0.00000,C 180.00000} ; retreat
  ; Step 2979, bar 1267
  LIN {X 985.893,Y -2029.899,Z 855.478,A 89.96659,B 0.00000,C 180.00000} ; outside
  LIN {X 985.893,Y -2029.899,Z -132.531,A 89.96659,B 0.00000,C 180.00000} ; preinsert
  LIN {X 985.893,Y -2029.899,Z -382.531,A 89.96659,B 0.00000,C 180.00000} ; insert
  LIN {X 985.893,Y -2029.899,Z -382.531,A 89.96659,B 0.00000,C 180.00000} ; release
  LIN {X 985.893,Y -2029.899,Z -82.531,A 89.96659,B 0.00000,C 180.00000} ; retreat
  ; Step 2980, bar 1269
  LIN {X 1110.893,Y -2029.899,Z 855.478,A 89.96659,B 0.00000,C 180.00000} ; outside
  LIN {X 1110.893,Y -2029.899,Z -132.531,A 89.96659,B 0.00000,C 180.00000} ; preinsert
  LIN {X 1110.893,Y -2029.899,Z -382.531,A 89.96659,B 0.00000,C 180.00000} ; insert
  LIN {X 1110.893,Y -2029.899,Z -382.531,A 89.96659,B 0.00000,C 180.00000} ; release
  LIN {X 1110.893,Y -2029.899,Z -82.531,A 89.96659,B 0.00000,C 180.00000} ; retreat
  ; Step 2981, bar 1271
  LIN {X 1235.893,Y -2029.899,Z 855.478,A 89.96659,B 0.00000,C 180.00000} ; outside
  LIN {X 1235.893,Y -2029.899,Z -132.531,A 89.96659,B 0.00000,C 180.00000} ; preinsert
  LIN {X 1235.893,Y -2029.899,Z -382.531,A 89.96659,B 0.00000,C 180.00000} ; insert
  LIN {X 1235.893,Y -2029.899,Z -382.531,A 89.96659,B 0.00000,C 180.00000} ; release
  LIN {X 1235.893,Y -2029.899,Z -82.531,A 89.96659,B 0.00000,C 180.00000} ; retreat
  ; Step 2982, bar 1273
  LIN {X 1360.893,Y -2029.899,Z 855.478,A 89.96659,B 0.00000,C 180.00000} ; outside
  LIN {X 1360.893,Y -2029.899,Z -132.531,A 89.96659,B 0.00000,C 180.00000} ; preinsert
  LIN {X 1360.893,Y -2029.899,Z -382.531,A 89.96659,B 0.00000,C 180.00000} ; insert
  LIN {X 1360.893,Y -2029.899,Z -382.531,A 89.96659,B 0.00000,C 180.00000} ; release
  LIN {X 1360.893,Y -2029.899,Z -82.531,A 89.96659,B 0.00000,C 180.00000} ; retreat
  ; Step 2983, bar 1275
  LIN {X 1485.893,Y -2029.899,Z 855.478,A 89.96659,B 0.00000,C 180.00000} ; outside
  LIN {X 1485.893,Y -2029.899,Z -132.531,A 89.96659,B 0.00000,C 180.00000} ; preinsert
  LIN {X 1485.893,Y -2029.899,Z -382.531,A 89.96659,B 0.00000,C 180.00000} ; insert
  LIN {X 1485.893,Y -2029.899,Z -382.531,A 89.96659,B 0.00000,C 180.00000} ; release
  LIN {X 1485.893,Y -2029.899,Z -82.531,A 89.96659,B 0.00000,C 180.00000} ; retreat
  ; Step 2984, bar 1277
  LIN {X 1610.893,Y -2029.899,Z 855.478,A 89.96659,B 0.00000,C 180.00000} ; outside
  LIN {X 1610.893,Y -2029.899,Z -132.531,A 89.96659,B 0.00000,C 180.00000} ; preinsert
  LIN {X 1610.893,Y -2029.899,Z -382.531,A 89.96659,B 0.00000,C 180.00000} ; insert
  LIN {X 1610.893,Y -2029.899,Z -382.531,A 89.96659,B 0.00000,C 180.00000} ; release
  LIN {X 1610.893,Y -2029.899,Z -82.531,A 89.96659,B 0.00000,C 180.00000} ; retreat
  ; Step 2985, bar 1279
  LIN {X 1735.893,Y -2029.899,Z 855.478,A 89.96659,B 0.00000,C 180.00000} ; outside
  LIN {X 1735.893,Y -2029.899,Z -132.531,A 89.96659,B 0.00000,C 180.00000} ; preinsert
  LIN {X 1735.893,Y -2029.899,Z -382.531,A 89.96659,B 0.00000,C 180.00000} ; insert
  LIN {X 1735.893,Y -2029.899,Z -382.531,A 89.96659,B 0.00000,C 180.00000} ; release
  LIN {X 1735.893,Y -2029.899,Z -82.531,A 89.96659,B 0.00000,C 180.00000} ; retreat
  ; Step 2986, bar 1281
  LIN {X 1860.893,Y -2029.899,Z 855.478,A 89.96659,B 0.00000,C 180.00000} ; outside
  LIN {X 1860.893,Y -2029.899,Z -132.531,A 89.96659,B 0.00000,C 180.00000} ; preinsert
  LIN {X 1860.893,Y -2029.899,Z -382.531,A 89.96659,B 0.00000,C 180.00000} ; insert
  LIN {X 1860.893,Y -2029.899,Z -382.531,A 89.96659,B 0.00000,C 180.00000} ; release
  LIN {X 1860.893,Y -2029.899,Z -82.531,A 89.96659,B 0.00000,C 180.00000} ; retreat
  ; Step 2987, bar 1283
  LIN {X 2110.893,Y -2029.899,Z 855.478,A 89.96659,B 0.00000,C 180.00000} ; outside
  LIN {X 2110.893,Y -2029.899,Z -132.531,A 89.96659,B 0.00000,C 180.00000} ; preinsert
  LIN {X 2110.893,Y -2029.899,Z -382.531,A 89.96659,B 0.00000,C 180.00000} ; insert
  LIN {X 2110.893,Y -2029.899,Z -382.531,A 89.96659,B 0.00000,C 180.00000} ; release
  LIN {X 2110.893,Y -2029.899,Z -82.531,A 89.96659,B 0.00000,C 180.00000} ; retreat
  ; Step 2988, bar 1285
  LIN {X 2235.893,Y -2029.899,Z 855.478,A 89.96659,B 0.00000,C 180.00000} ; outside
  LIN {X 2235.893,Y -2029.899,Z -132.531,A 89.96659,B 0.00000,C 180.00000} ; preinsert
  LIN {X 2235.893,Y -2029.899,Z -382.531,A 89.96659,B 0.00000,C 180.00000} ; insert
  LIN {X 2235.893,Y -2029.899,Z -382.531,A 89.96659,B 0.00000,C 180.00000} ; release
  LIN {X 2235.893,Y -2029.899,Z -82.531,A 89.96659,B 0.00000,C 180.00000} ; retreat
  ; Step 2989, bar 1287
  LIN {X 2360.893,Y -2029.899,Z 855.478,A 89.96659,B 0.00000,C 180.00000} ; outside
  LIN {X 2360.893,Y -2029.899,Z -132.531,A 89.96659,B 0.00000,C 180.00000} ; preinsert
  LIN {X 2360.893,Y -2029.899,Z -382.531,A 89.96659,B 0.00000,C 180.00000} ; insert
  LIN {X 2360.893,Y -2029.899,Z -382.531,A 89.96659,B 0.00000,C 180.00000} ; release
  LIN {X 2360.893,Y -2029.899,Z -82.531,A 89.96659,B 0.00000,C 180.00000} ; retreat
  ; Step 2990, bar 1289
  LIN {X 2485.893,Y -2029.899,Z 855.478,A 89.96659,B 0.00000,C 180.00000} ; outside
  LIN {X 2485.893,Y -2029.899,Z -132.531,A 89.96659,B 0.00000,C 180.00000} ; preinsert
  LIN {X 2485.893,Y -2029.899,Z -382.531,A 89.96659,B 0.00000,C 180.00000} ; insert
  LIN {X 2485.893,Y -2029.899,Z -382.531,A 89.96659,B 0.00000,C 180.00000} ; release
  LIN {X 2485.893,Y -2029.899,Z -82.531,A 89.96659,B 0.00000,C 180.00000} ; retreat
  ; Step 2991, bar 1291
  LIN {X 2610.893,Y -2029.899,Z 855.478,A 89.96659,B 0.00000,C 180.00000} ; outside
  LIN {X 2610.893,Y -2029.899,Z -132.531,A 89.96659,B 0.00000,C 180.00000} ; preinsert
  LIN {X 2610.893,Y -2029.899,Z -382.531,A 89.96659,B 0.00000,C 180.00000} ; insert
  LIN {X 2610.893,Y -2029.899,Z -382.531,A 89.96659,B 0.00000,C 180.00000} ; release
  LIN {X 2610.893,Y -2029.899,Z -82.531,A 89.96659,B 0.00000,C 180.00000} ; retreat
  ; Step 2992, bar 1293
  LIN {X 2735.893,Y -2029.899,Z 855.478,A 89.96659,B 0.00000,C 180.00000} ; outside
  LIN {X 2735.893,Y -2029.899,Z -132.531,A 89.96659,B 0.00000,C 180.00000} ; preinsert
  LIN {X 2735.893,Y -2029.899,Z -382.531,A 89.96659,B 0.00000,C 180.00000} ; insert
  LIN {X 2735.893,Y -2029.899,Z -382.531,A 89.96659,B 0.00000,C 180.00000} ; release
  LIN {X 2735.893,Y -2029.899,Z -82.531,A 89.96659,B 0.00000,C 180.00000} ; retreat
  ; Step 2993, bar 1295
  LIN {X 2860.893,Y -2029.899,Z 855.478,A 89.96659,B 0.00000,C 180.00000} ; outside
  LIN {X 2860.893,Y -2029.899,Z -132.531,A 89.96659,B 0.00000,C 180.00000} ; preinsert
  LIN {X 2860.893,Y -2029.899,Z -382.531,A 89.96659,B 0.00000,C 180.00000} ; insert
  LIN {X 2860.893,Y -2029.899,Z -382.531,A 89.96659,B 0.00000,C 180.00000} ; release
  LIN {X 2860.893,Y -2029.899,Z -82.531,A 89.96659,B 0.00000,C 180.00000} ; retreat
  ; Step 2994, bar 1297
  LIN {X 2985.893,Y -2029.899,Z 855.478,A 89.96659,B 0.00000,C 180.00000} ; outside
  LIN {X 2985.893,Y -2029.899,Z -132.531,A 89.96659,B 0.00000,C 180.00000} ; preinsert
  LIN {X 2985.893,Y -2029.899,Z -382.531,A 89.96659,B 0.00000,C 180.00000} ; insert
  LIN {X 2985.893,Y -2029.899,Z -382.531,A 89.96659,B 0.00000,C 180.00000} ; release
  LIN {X 2985.893,Y -2029.899,Z -82.531,A 89.96659,B 0.00000,C 180.00000} ; retreat
  ; Step 2995, bar 1299
  LIN {X 3110.893,Y -2029.899,Z 855.478,A 89.96659,B 0.00000,C 180.00000} ; outside
  LIN {X 3110.893,Y -2029.899,Z -132.531,A 89.96659,B 0.00000,C 180.00000} ; preinsert
  LIN {X 3110.893,Y -2029.899,Z -382.531,A 89.96659,B 0.00000,C 180.00000} ; insert
  LIN {X 3110.893,Y -2029.899,Z -382.531,A 89.96659,B 0.00000,C 180.00000} ; release
  LIN {X 3110.893,Y -2029.899,Z -82.531,A 89.96659,B 0.00000,C 180.00000} ; retreat
  ; Step 2996, bar 1301
  LIN {X 3235.893,Y -2029.899,Z 855.478,A 89.96659,B 0.00000,C 180.00000} ; outside
  LIN {X 3235.893,Y -2029.899,Z -132.531,A 89.96659,B 0.00000,C 180.00000} ; preinsert
  LIN {X 3235.893,Y -2029.899,Z -382.531,A 89.96659,B 0.00000,C 180.00000} ; insert
  LIN {X 3235.893,Y -2029.899,Z -382.531,A 89.96659,B 0.00000,C 180.00000} ; release
  LIN {X 3235.893,Y -2029.899,Z -82.531,A 89.96659,B 0.00000,C 180.00000} ; retreat
  ; Step 2997, bar 1303
  LIN {X 3360.893,Y -2029.899,Z 855.478,A 89.96659,B 0.00000,C 180.00000} ; outside
  LIN {X 3360.893,Y -2029.899,Z -132.531,A 89.96659,B 0.00000,C 180.00000} ; preinsert
  LIN {X 3360.893,Y -2029.899,Z -382.531,A 89.96659,B 0.00000,C 180.00000} ; insert
  LIN {X 3360.893,Y -2029.899,Z -382.531,A 89.96659,B 0.00000,C 180.00000} ; release
  LIN {X 3360.893,Y -2029.899,Z -82.531,A 89.96659,B 0.00000,C 180.00000} ; retreat
  ; Step 2998, bar 1305
  LIN {X 3485.893,Y -2029.899,Z 855.478,A 89.96659,B 0.00000,C 180.00000} ; outside
  LIN {X 3485.893,Y -2029.899,Z -132.531,A 89.96659,B 0.00000,C 180.00000} ; preinsert
  LIN {X 3485.893,Y -2029.899,Z -382.531,A 89.96659,B 0.00000,C 180.00000} ; insert
  LIN {X 3485.893,Y -2029.899,Z -382.531,A 89.96659,B 0.00000,C 180.00000} ; release
  LIN {X 3485.893,Y -2029.899,Z -82.531,A 89.96659,B 0.00000,C 180.00000} ; retreat
  ; Step 2999, bar 1307
  LIN {X 3610.893,Y -2029.899,Z 855.478,A 89.96659,B 0.00000,C 180.00000} ; outside
  LIN {X 3610.893,Y -2029.899,Z -132.531,A 89.96659,B 0.00000,C 180.00000} ; preinsert
  LIN {X 3610.893,Y -2029.899,Z -382.531,A 89.96659,B 0.00000,C 180.00000} ; insert
  LIN {X 3610.893,Y -2029.899,Z -382.531,A 89.96659,B 0.00000,C 180.00000} ; release
  LIN {X 3610.893,Y -2029.899,Z -82.531,A 89.96659,B 0.00000,C 180.00000} ; retreat
  ; Step 3000, bar 1309
  LIN {X 3735.893,Y -2029.899,Z 855.478,A 89.96659,B 0.00000,C 180.00000} ; outside
  LIN {X 3735.893,Y -2029.899,Z -132.531,A 89.96659,B 0.00000,C 180.00000} ; preinsert
  LIN {X 3735.893,Y -2029.899,Z -382.531,A 89.96659,B 0.00000,C 180.00000} ; insert
  LIN {X 3735.893,Y -2029.899,Z -382.531,A 89.96659,B 0.00000,C 180.00000} ; release
  LIN {X 3735.893,Y -2029.899,Z -82.531,A 89.96659,B 0.00000,C 180.00000} ; retreat
  ; Step 3001, bar 1311
  LIN {X 3860.893,Y -2029.899,Z 855.478,A 89.96659,B 0.00000,C 180.00000} ; outside
  LIN {X 3860.893,Y -2029.899,Z -132.531,A 89.96659,B 0.00000,C 180.00000} ; preinsert
  LIN {X 3860.893,Y -2029.899,Z -382.531,A 89.96659,B 0.00000,C 180.00000} ; insert
  LIN {X 3860.893,Y -2029.899,Z -382.531,A 89.96659,B 0.00000,C 180.00000} ; release
  LIN {X 3860.893,Y -2029.899,Z -82.531,A 89.96659,B 0.00000,C 180.00000} ; retreat
  ; Step 3002, bar 1313
  LIN {X 3985.893,Y -2029.899,Z 855.478,A 89.96659,B 0.00000,C 180.00000} ; outside
  LIN {X 3985.893,Y -2029.899,Z -132.531,A 89.96659,B 0.00000,C 180.00000} ; preinsert
  LIN {X 3985.893,Y -2029.899,Z -382.531,A 89.96659,B 0.00000,C 180.00000} ; insert
  LIN {X 3985.893,Y -2029.899,Z -382.531,A 89.96659,B 0.00000,C 180.00000} ; release
  LIN {X 3985.893,Y -2029.899,Z -82.531,A 89.96659,B 0.00000,C 180.00000} ; retreat
  ; Step 3003, bar 1315
  LIN {X 4110.893,Y -2029.899,Z 855.478,A 89.96659,B 0.00000,C -180.00000} ; outside
  LIN {X 4110.893,Y -2029.899,Z -132.531,A 89.96659,B 0.00000,C -180.00000} ; preinsert
  LIN {X 4110.893,Y -2029.899,Z -382.531,A 89.96659,B 0.00000,C -180.00000} ; insert
  LIN {X 4110.893,Y -2029.899,Z -382.531,A 89.96659,B 0.00000,C -180.00000} ; release
  LIN {X 4110.893,Y -2029.899,Z -82.531,A 89.96659,B 0.00000,C -180.00000} ; retreat
  ; Step 3004, bar 1317
  LIN {X 4235.893,Y -2029.899,Z 855.478,A 89.96659,B 0.00000,C -180.00000} ; outside
  LIN {X 4235.893,Y -2029.899,Z -132.531,A 89.96659,B 0.00000,C -180.00000} ; preinsert
  LIN {X 4235.893,Y -2029.899,Z -382.531,A 89.96659,B 0.00000,C -180.00000} ; insert
  LIN {X 4235.893,Y -2029.899,Z -382.531,A 89.96659,B 0.00000,C -180.00000} ; release
  LIN {X 4235.893,Y -2029.899,Z -82.531,A 89.96659,B 0.00000,C -180.00000} ; retreat
  ; Step 3005, bar 1319
  LIN {X 4360.893,Y -2029.899,Z 855.478,A 89.96659,B 0.00000,C -180.00000} ; outside
  LIN {X 4360.893,Y -2029.899,Z -132.531,A 89.96659,B 0.00000,C -180.00000} ; preinsert
  LIN {X 4360.893,Y -2029.899,Z -382.531,A 89.96659,B 0.00000,C -180.00000} ; insert
  LIN {X 4360.893,Y -2029.899,Z -382.531,A 89.96659,B 0.00000,C -180.00000} ; release
  LIN {X 4360.893,Y -2029.899,Z -82.531,A 89.96659,B 0.00000,C -180.00000} ; retreat
  ; Step 3006, bar 1321
  LIN {X 4485.893,Y -2029.899,Z 855.478,A 89.96659,B 0.00000,C -180.00000} ; outside
  LIN {X 4485.893,Y -2029.899,Z -132.531,A 89.96659,B 0.00000,C -180.00000} ; preinsert
  LIN {X 4485.893,Y -2029.899,Z -382.531,A 89.96659,B 0.00000,C -180.00000} ; insert
  LIN {X 4485.893,Y -2029.899,Z -382.531,A 89.96659,B 0.00000,C -180.00000} ; release
  LIN {X 4485.893,Y -2029.899,Z -82.531,A 89.96659,B 0.00000,C -180.00000} ; retreat
  ; Step 3007, bar 1323
  LIN {X 4610.893,Y -2029.899,Z 855.478,A 89.96659,B 0.00000,C -180.00000} ; outside
  LIN {X 4610.893,Y -2029.899,Z -132.531,A 89.96659,B 0.00000,C -180.00000} ; preinsert
  LIN {X 4610.893,Y -2029.899,Z -382.531,A 89.96659,B 0.00000,C -180.00000} ; insert
  LIN {X 4610.893,Y -2029.899,Z -382.531,A 89.96659,B 0.00000,C -180.00000} ; release
  LIN {X 4610.893,Y -2029.899,Z -82.531,A 89.96659,B 0.00000,C -180.00000} ; retreat
  ; Step 3008, bar 1325
  LIN {X 4735.893,Y -2029.899,Z 855.478,A 89.96659,B 0.00000,C -180.00000} ; outside
  LIN {X 4735.893,Y -2029.899,Z -132.531,A 89.96659,B 0.00000,C -180.00000} ; preinsert
  LIN {X 4735.893,Y -2029.899,Z -382.531,A 89.96659,B 0.00000,C -180.00000} ; insert
  LIN {X 4735.893,Y -2029.899,Z -382.531,A 89.96659,B 0.00000,C -180.00000} ; release
  LIN {X 4735.893,Y -2029.899,Z -82.531,A 89.96659,B 0.00000,C -180.00000} ; retreat
  ; Step 3009, bar 1327
  LIN {X 4860.893,Y -2029.899,Z 855.478,A 89.96659,B 0.00000,C -180.00000} ; outside
  LIN {X 4860.893,Y -2029.899,Z -132.531,A 89.96659,B 0.00000,C -180.00000} ; preinsert
  LIN {X 4860.893,Y -2029.899,Z -382.531,A 89.96659,B 0.00000,C -180.00000} ; insert
  LIN {X 4860.893,Y -2029.899,Z -382.531,A 89.96659,B 0.00000,C -180.00000} ; release
  LIN {X 4860.893,Y -2029.899,Z -82.531,A 89.96659,B 0.00000,C -180.00000} ; retreat
  ; Step 3010, bar 1329
  LIN {X 4985.893,Y -2029.899,Z 855.478,A 89.96659,B 0.00000,C -180.00000} ; outside
  LIN {X 4985.893,Y -2029.899,Z -132.531,A 89.96659,B 0.00000,C -180.00000} ; preinsert
  LIN {X 4985.893,Y -2029.899,Z -382.531,A 89.96659,B 0.00000,C -180.00000} ; insert
  LIN {X 4985.893,Y -2029.899,Z -382.531,A 89.96659,B 0.00000,C -180.00000} ; release
  LIN {X 4985.893,Y -2029.899,Z -82.531,A 89.96659,B 0.00000,C -180.00000} ; retreat
  ; Step 3011, bar 1331
  LIN {X 5110.893,Y -2029.899,Z 855.478,A 89.96659,B 0.00000,C -180.00000} ; outside
  LIN {X 5110.893,Y -2029.899,Z -132.531,A 89.96659,B 0.00000,C -180.00000} ; preinsert
  LIN {X 5110.893,Y -2029.899,Z -382.531,A 89.96659,B 0.00000,C -180.00000} ; insert
  LIN {X 5110.893,Y -2029.899,Z -382.531,A 89.96659,B 0.00000,C -180.00000} ; release
  LIN {X 5110.893,Y -2029.899,Z -82.531,A 89.96659,B 0.00000,C -180.00000} ; retreat
  ; Step 3012, bar 1333
  LIN {X 5235.893,Y -2029.899,Z 855.478,A 89.96659,B 0.00000,C -180.00000} ; outside
  LIN {X 5235.893,Y -2029.899,Z -132.531,A 89.96659,B 0.00000,C -180.00000} ; preinsert
  LIN {X 5235.893,Y -2029.899,Z -382.531,A 89.96659,B 0.00000,C -180.00000} ; insert
  LIN {X 5235.893,Y -2029.899,Z -382.531,A 89.96659,B 0.00000,C -180.00000} ; release
  LIN {X 5235.893,Y -2029.899,Z -82.531,A 89.96659,B 0.00000,C -180.00000} ; retreat
  ; Step 3013, bar 1335
  LIN {X 5360.893,Y -2029.899,Z 855.478,A 89.96659,B 0.00000,C -180.00000} ; outside
  LIN {X 5360.893,Y -2029.899,Z -132.531,A 89.96659,B 0.00000,C -180.00000} ; preinsert
  LIN {X 5360.893,Y -2029.899,Z -382.531,A 89.96659,B 0.00000,C -180.00000} ; insert
  LIN {X 5360.893,Y -2029.899,Z -382.531,A 89.96659,B 0.00000,C -180.00000} ; release
  LIN {X 5360.893,Y -2029.899,Z -82.531,A 89.96659,B 0.00000,C -180.00000} ; retreat
  ; Step 3014, bar 1337
  LIN {X 5485.893,Y -2029.899,Z 855.478,A 89.96659,B 0.00000,C -180.00000} ; outside
  LIN {X 5485.893,Y -2029.899,Z -132.531,A 89.96659,B 0.00000,C -180.00000} ; preinsert
  LIN {X 5485.893,Y -2029.899,Z -382.531,A 89.96659,B 0.00000,C -180.00000} ; insert
  LIN {X 5485.893,Y -2029.899,Z -382.531,A 89.96659,B 0.00000,C -180.00000} ; release
  LIN {X 5485.893,Y -2029.899,Z -82.531,A 89.96659,B 0.00000,C -180.00000} ; retreat
  ; Step 3015, bar 1339
  LIN {X 5610.893,Y -2029.899,Z 855.478,A 89.96659,B 0.00000,C -180.00000} ; outside
  LIN {X 5610.893,Y -2029.899,Z -132.531,A 89.96659,B 0.00000,C -180.00000} ; preinsert
  LIN {X 5610.893,Y -2029.899,Z -382.531,A 89.96659,B 0.00000,C -180.00000} ; insert
  LIN {X 5610.893,Y -2029.899,Z -382.531,A 89.96659,B 0.00000,C -180.00000} ; release
  LIN {X 5610.893,Y -2029.899,Z -82.531,A 89.96659,B 0.00000,C -180.00000} ; retreat
  ; Step 3016, bar 1341
  LIN {X 5735.893,Y -2029.899,Z 855.478,A 89.96659,B 0.00000,C -180.00000} ; outside
  LIN {X 5735.893,Y -2029.899,Z -132.531,A 89.96659,B 0.00000,C -180.00000} ; preinsert
  LIN {X 5735.893,Y -2029.899,Z -382.531,A 89.96659,B 0.00000,C -180.00000} ; insert
  LIN {X 5735.893,Y -2029.899,Z -382.531,A 89.96659,B 0.00000,C -180.00000} ; release
  LIN {X 5735.893,Y -2029.899,Z -82.531,A 89.96659,B 0.00000,C -180.00000} ; retreat
  ; Step 3017, bar 1343
  LIN {X 5860.893,Y -2029.899,Z 855.478,A 89.96659,B 0.00000,C -180.00000} ; outside
  LIN {X 5860.893,Y -2029.899,Z -132.531,A 89.96659,B 0.00000,C -180.00000} ; preinsert
  LIN {X 5860.893,Y -2029.899,Z -382.531,A 89.96659,B 0.00000,C -180.00000} ; insert
  LIN {X 5860.893,Y -2029.899,Z -382.531,A 89.96659,B 0.00000,C -180.00000} ; release
  LIN {X 5860.893,Y -2029.899,Z -82.531,A 89.96659,B 0.00000,C -180.00000} ; retreat
  ; Step 3018, bar 1345
  LIN {X 6110.893,Y -2029.899,Z 855.478,A 89.96659,B 0.00000,C -180.00000} ; outside
  LIN {X 6110.893,Y -2029.899,Z -132.531,A 89.96659,B 0.00000,C -180.00000} ; preinsert
  LIN {X 6110.893,Y -2029.899,Z -382.531,A 89.96659,B 0.00000,C -180.00000} ; insert
  LIN {X 6110.893,Y -2029.899,Z -382.531,A 89.96659,B 0.00000,C -180.00000} ; release
  LIN {X 6110.893,Y -2029.899,Z -82.531,A 89.96659,B 0.00000,C -180.00000} ; retreat
  ; Step 3019, bar 1347
  LIN {X 6235.893,Y -2029.899,Z 855.478,A 89.96659,B 0.00000,C -180.00000} ; outside
  LIN {X 6235.893,Y -2029.899,Z -132.531,A 89.96659,B 0.00000,C -180.00000} ; preinsert
  LIN {X 6235.893,Y -2029.899,Z -382.531,A 89.96659,B 0.00000,C -180.00000} ; insert
  LIN {X 6235.893,Y -2029.899,Z -382.531,A 89.96659,B 0.00000,C -180.00000} ; release
  LIN {X 6235.893,Y -2029.899,Z -82.531,A 89.96659,B 0.00000,C -180.00000} ; retreat
  ; Step 3020, bar 1349
  LIN {X 6360.893,Y -2029.899,Z 855.478,A 89.96659,B 0.00000,C -180.00000} ; outside
  LIN {X 6360.893,Y -2029.899,Z -132.531,A 89.96659,B 0.00000,C -180.00000} ; preinsert
  LIN {X 6360.893,Y -2029.899,Z -382.531,A 89.96659,B 0.00000,C -180.00000} ; insert
  LIN {X 6360.893,Y -2029.899,Z -382.531,A 89.96659,B 0.00000,C -180.00000} ; release
  LIN {X 6360.893,Y -2029.899,Z -82.531,A 89.96659,B 0.00000,C -180.00000} ; retreat
  ; Step 3021, bar 1351
  LIN {X 6485.893,Y -2029.899,Z 855.478,A 89.96659,B 0.00000,C -180.00000} ; outside
  LIN {X 6485.893,Y -2029.899,Z -132.531,A 89.96659,B 0.00000,C -180.00000} ; preinsert
  LIN {X 6485.893,Y -2029.899,Z -382.531,A 89.96659,B 0.00000,C -180.00000} ; insert
  LIN {X 6485.893,Y -2029.899,Z -382.531,A 89.96659,B 0.00000,C -180.00000} ; release
  LIN {X 6485.893,Y -2029.899,Z -82.531,A 89.96659,B 0.00000,C -180.00000} ; retreat
  ; Step 3022, bar 1353
  LIN {X 6610.893,Y -2029.899,Z 855.478,A 89.96659,B 0.00000,C -180.00000} ; outside
  LIN {X 6610.893,Y -2029.899,Z -132.531,A 89.96659,B 0.00000,C -180.00000} ; preinsert
  LIN {X 6610.893,Y -2029.899,Z -382.531,A 89.96659,B 0.00000,C -180.00000} ; insert
  LIN {X 6610.893,Y -2029.899,Z -382.531,A 89.96659,B 0.00000,C -180.00000} ; release
  LIN {X 6610.893,Y -2029.899,Z -82.531,A 89.96659,B 0.00000,C -180.00000} ; retreat
  ; Step 3023, bar 1355
  LIN {X 6735.893,Y -2029.899,Z 855.478,A 89.96659,B 0.00000,C -180.00000} ; outside
  LIN {X 6735.893,Y -2029.899,Z -132.531,A 89.96659,B 0.00000,C -180.00000} ; preinsert
  LIN {X 6735.893,Y -2029.899,Z -382.531,A 89.96659,B 0.00000,C -180.00000} ; insert
  LIN {X 6735.893,Y -2029.899,Z -382.531,A 89.96659,B 0.00000,C -180.00000} ; release
  LIN {X 6735.893,Y -2029.899,Z -82.531,A 89.96659,B 0.00000,C -180.00000} ; retreat
  ; Step 3024, bar 1357
  LIN {X 6860.893,Y -2029.899,Z 855.478,A 89.96659,B 0.00000,C -180.00000} ; outside
  LIN {X 6860.893,Y -2029.899,Z -132.531,A 89.96659,B 0.00000,C -180.00000} ; preinsert
  LIN {X 6860.893,Y -2029.899,Z -382.531,A 89.96659,B 0.00000,C -180.00000} ; insert
  LIN {X 6860.893,Y -2029.899,Z -382.531,A 89.96659,B 0.00000,C -180.00000} ; release
  LIN {X 6860.893,Y -2029.899,Z -82.531,A 89.96659,B 0.00000,C -180.00000} ; retreat
  ; Step 3025, bar 1359
  LIN {X 6985.893,Y -2029.899,Z 855.478,A 89.96659,B 0.00000,C -180.00000} ; outside
  LIN {X 6985.893,Y -2029.899,Z -132.531,A 89.96659,B 0.00000,C -180.00000} ; preinsert
  LIN {X 6985.893,Y -2029.899,Z -382.531,A 89.96659,B 0.00000,C -180.00000} ; insert
  LIN {X 6985.893,Y -2029.899,Z -382.531,A 89.96659,B 0.00000,C -180.00000} ; release
  LIN {X 6985.893,Y -2029.899,Z -82.531,A 89.96659,B 0.00000,C -180.00000} ; retreat
  ; Step 3026, bar 1361
  LIN {X 7110.893,Y -2029.899,Z 855.478,A 89.96659,B 0.00000,C -180.00000} ; outside
  LIN {X 7110.893,Y -2029.899,Z -132.531,A 89.96659,B 0.00000,C -180.00000} ; preinsert
  LIN {X 7110.893,Y -2029.899,Z -382.531,A 89.96659,B 0.00000,C -180.00000} ; insert
  LIN {X 7110.893,Y -2029.899,Z -382.531,A 89.96659,B 0.00000,C -180.00000} ; release
  LIN {X 7110.893,Y -2029.899,Z -82.531,A 89.96659,B 0.00000,C -180.00000} ; retreat
  ; Step 3027, bar 1363
  LIN {X 7235.893,Y -2029.899,Z 855.478,A 89.96659,B 0.00000,C -180.00000} ; outside
  LIN {X 7235.893,Y -2029.899,Z -132.531,A 89.96659,B 0.00000,C -180.00000} ; preinsert
  LIN {X 7235.893,Y -2029.899,Z -382.531,A 89.96659,B 0.00000,C -180.00000} ; insert
  LIN {X 7235.893,Y -2029.899,Z -382.531,A 89.96659,B 0.00000,C -180.00000} ; release
  LIN {X 7235.893,Y -2029.899,Z -82.531,A 89.96659,B 0.00000,C -180.00000} ; retreat
  ; Step 3028, bar 1365
  LIN {X 7360.893,Y -2029.899,Z 855.478,A 89.96659,B 0.00000,C -180.00000} ; outside
  LIN {X 7360.893,Y -2029.899,Z -132.531,A 89.96659,B 0.00000,C -180.00000} ; preinsert
  LIN {X 7360.893,Y -2029.899,Z -382.531,A 89.96659,B 0.00000,C -180.00000} ; insert
  LIN {X 7360.893,Y -2029.899,Z -382.531,A 89.96659,B 0.00000,C -180.00000} ; release
  LIN {X 7360.893,Y -2029.899,Z -82.531,A 89.96659,B 0.00000,C -180.00000} ; retreat
  ; Step 3029, bar 1367
  LIN {X 7485.893,Y -2029.899,Z 855.478,A 89.96659,B 0.00000,C -180.00000} ; outside
  LIN {X 7485.893,Y -2029.899,Z -132.531,A 89.96659,B 0.00000,C -180.00000} ; preinsert
  LIN {X 7485.893,Y -2029.899,Z -382.531,A 89.96659,B 0.00000,C -180.00000} ; insert
  LIN {X 7485.893,Y -2029.899,Z -382.531,A 89.96659,B 0.00000,C -180.00000} ; release
  LIN {X 7485.893,Y -2029.899,Z -82.531,A 89.96659,B 0.00000,C -180.00000} ; retreat
  ; Step 3030, bar 1369
  LIN {X 7610.893,Y -2029.899,Z 855.478,A 89.96659,B 0.00000,C -180.00000} ; outside
  LIN {X 7610.893,Y -2029.899,Z -132.531,A 89.96659,B 0.00000,C -180.00000} ; preinsert
  LIN {X 7610.893,Y -2029.899,Z -382.531,A 89.96659,B 0.00000,C -180.00000} ; insert
  LIN {X 7610.893,Y -2029.899,Z -382.531,A 89.96659,B 0.00000,C -180.00000} ; release
  LIN {X 7610.893,Y -2029.899,Z -82.531,A 89.96659,B 0.00000,C -180.00000} ; retreat
  ; Step 3031, bar 1371
  LIN {X 7735.893,Y -2029.899,Z 855.478,A 89.96659,B 0.00000,C -180.00000} ; outside
  LIN {X 7735.893,Y -2029.899,Z -132.531,A 89.96659,B 0.00000,C -180.00000} ; preinsert
  LIN {X 7735.893,Y -2029.899,Z -382.531,A 89.96659,B 0.00000,C -180.00000} ; insert
  LIN {X 7735.893,Y -2029.899,Z -382.531,A 89.96659,B 0.00000,C -180.00000} ; release
  LIN {X 7735.893,Y -2029.899,Z -82.531,A 89.96659,B 0.00000,C -180.00000} ; retreat
  ; Step 3032, bar 1373
  LIN {X 7860.893,Y -2029.899,Z 855.478,A 89.96659,B 0.00000,C -180.00000} ; outside
  LIN {X 7860.893,Y -2029.899,Z -132.531,A 89.96659,B 0.00000,C -180.00000} ; preinsert
  LIN {X 7860.893,Y -2029.899,Z -382.531,A 89.96659,B 0.00000,C -180.00000} ; insert
  LIN {X 7860.893,Y -2029.899,Z -382.531,A 89.96659,B 0.00000,C -180.00000} ; release
  LIN {X 7860.893,Y -2029.899,Z -82.531,A 89.96659,B 0.00000,C -180.00000} ; retreat
  ; Step 3033, bar 1375
  LIN {X 7985.893,Y -2029.899,Z 855.478,A 89.96659,B 0.00000,C -180.00000} ; outside
  LIN {X 7985.893,Y -2029.899,Z -132.531,A 89.96659,B 0.00000,C -180.00000} ; preinsert
  LIN {X 7985.893,Y -2029.899,Z -382.531,A 89.96659,B 0.00000,C -180.00000} ; insert
  LIN {X 7985.893,Y -2029.899,Z -382.531,A 89.96659,B 0.00000,C -180.00000} ; release
  LIN {X 7985.893,Y -2029.899,Z -82.531,A 89.96659,B 0.00000,C -180.00000} ; retreat
  ; Step 3034, bar 1377
  LIN {X 8110.893,Y -2029.899,Z 855.478,A 89.96659,B 0.00000,C -180.00000} ; outside
  LIN {X 8110.893,Y -2029.899,Z -132.531,A 89.96659,B 0.00000,C -180.00000} ; preinsert
  LIN {X 8110.893,Y -2029.899,Z -382.531,A 89.96659,B 0.00000,C -180.00000} ; insert
  LIN {X 8110.893,Y -2029.899,Z -382.531,A 89.96659,B 0.00000,C -180.00000} ; release
  LIN {X 8110.893,Y -2029.899,Z -82.531,A 89.96659,B 0.00000,C -180.00000} ; retreat
  ; Step 3035, bar 1379
  LIN {X 8235.893,Y -2029.899,Z 855.478,A 89.96659,B 0.00000,C 180.00000} ; outside
  LIN {X 8235.893,Y -2029.899,Z -132.531,A 89.96659,B 0.00000,C 180.00000} ; preinsert
  LIN {X 8235.893,Y -2029.899,Z -382.531,A 89.96659,B 0.00000,C 180.00000} ; insert
  LIN {X 8235.893,Y -2029.899,Z -382.531,A 89.96659,B 0.00000,C 180.00000} ; release
  LIN {X 8235.893,Y -2029.899,Z -82.531,A 89.96659,B 0.00000,C 180.00000} ; retreat
  ; Step 3036, bar 1381
  LIN {X 8360.893,Y -2029.899,Z 855.478,A 89.96659,B 0.00000,C 180.00000} ; outside
  LIN {X 8360.893,Y -2029.899,Z -132.531,A 89.96659,B 0.00000,C 180.00000} ; preinsert
  LIN {X 8360.893,Y -2029.899,Z -382.531,A 89.96659,B 0.00000,C 180.00000} ; insert
  LIN {X 8360.893,Y -2029.899,Z -382.531,A 89.96659,B 0.00000,C 180.00000} ; release
  LIN {X 8360.893,Y -2029.899,Z -82.531,A 89.96659,B 0.00000,C 180.00000} ; retreat
  ; Step 3037, bar 1383
  LIN {X 8485.893,Y -2029.899,Z 855.478,A 89.96659,B 0.00000,C 180.00000} ; outside
  LIN {X 8485.893,Y -2029.899,Z -132.531,A 89.96659,B 0.00000,C 180.00000} ; preinsert
  LIN {X 8485.893,Y -2029.899,Z -382.531,A 89.96659,B 0.00000,C 180.00000} ; insert
  LIN {X 8485.893,Y -2029.899,Z -382.531,A 89.96659,B 0.00000,C 180.00000} ; release
  LIN {X 8485.893,Y -2029.899,Z -82.531,A 89.96659,B 0.00000,C 180.00000} ; retreat
  ; Step 3038, bar 1385
  LIN {X 8610.893,Y -2029.899,Z 855.478,A 89.96659,B 0.00000,C 180.00000} ; outside
  LIN {X 8610.893,Y -2029.899,Z -132.531,A 89.96659,B 0.00000,C 180.00000} ; preinsert
  LIN {X 8610.893,Y -2029.899,Z -382.531,A 89.96659,B 0.00000,C 180.00000} ; insert
  LIN {X 8610.893,Y -2029.899,Z -382.531,A 89.96659,B 0.00000,C 180.00000} ; release
  LIN {X 8610.893,Y -2029.899,Z -82.531,A 89.96659,B 0.00000,C 180.00000} ; retreat
  ; Step 3039, bar 1387
  LIN {X 8735.893,Y -2029.899,Z 855.478,A 89.96659,B 0.00000,C 180.00000} ; outside
  LIN {X 8735.893,Y -2029.899,Z -132.531,A 89.96659,B 0.00000,C 180.00000} ; preinsert
  LIN {X 8735.893,Y -2029.899,Z -382.531,A 89.96659,B 0.00000,C 180.00000} ; insert
  LIN {X 8735.893,Y -2029.899,Z -382.531,A 89.96659,B 0.00000,C 180.00000} ; release
  LIN {X 8735.893,Y -2029.899,Z -82.531,A 89.96659,B 0.00000,C 180.00000} ; retreat
  ; Step 3040, bar 1389
  LIN {X 8860.893,Y -2029.899,Z 855.478,A 89.96659,B 0.00000,C 180.00000} ; outside
  LIN {X 8860.893,Y -2029.899,Z -132.531,A 89.96659,B 0.00000,C 180.00000} ; preinsert
  LIN {X 8860.893,Y -2029.899,Z -382.531,A 89.96659,B 0.00000,C 180.00000} ; insert
  LIN {X 8860.893,Y -2029.899,Z -382.531,A 89.96659,B 0.00000,C 180.00000} ; release
  LIN {X 8860.893,Y -2029.899,Z -82.531,A 89.96659,B 0.00000,C 180.00000} ; retreat
  ; Step 3041, bar 1391
  LIN {X 8985.893,Y -2029.899,Z 855.478,A 89.96659,B 0.00000,C 180.00000} ; outside
  LIN {X 8985.893,Y -2029.899,Z -132.531,A 89.96659,B 0.00000,C 180.00000} ; preinsert
  LIN {X 8985.893,Y -2029.899,Z -382.531,A 89.96659,B 0.00000,C 180.00000} ; insert
  LIN {X 8985.893,Y -2029.899,Z -382.531,A 89.96659,B 0.00000,C 180.00000} ; release
  LIN {X 8985.893,Y -2029.899,Z -82.531,A 89.96659,B 0.00000,C 180.00000} ; retreat
  ; Step 3042, bar 1393
  LIN {X 9110.893,Y -2029.899,Z 855.478,A 89.96659,B 0.00000,C 180.00000} ; outside
  LIN {X 9110.893,Y -2029.899,Z -132.531,A 89.96659,B 0.00000,C 180.00000} ; preinsert
  LIN {X 9110.893,Y -2029.899,Z -382.531,A 89.96659,B 0.00000,C 180.00000} ; insert
  LIN {X 9110.893,Y -2029.899,Z -382.531,A 89.96659,B 0.00000,C 180.00000} ; release
  LIN {X 9110.893,Y -2029.899,Z -82.531,A 89.96659,B 0.00000,C 180.00000} ; retreat
  ; Step 3043, bar 1395
  LIN {X 9235.893,Y -2029.899,Z 855.478,A 89.96659,B 0.00000,C 180.00000} ; outside
  LIN {X 9235.893,Y -2029.899,Z -132.531,A 89.96659,B 0.00000,C 180.00000} ; preinsert
  LIN {X 9235.893,Y -2029.899,Z -382.531,A 89.96659,B 0.00000,C 180.00000} ; insert
  LIN {X 9235.893,Y -2029.899,Z -382.531,A 89.96659,B 0.00000,C 180.00000} ; release
  LIN {X 9235.893,Y -2029.899,Z -82.531,A 89.96659,B 0.00000,C 180.00000} ; retreat
  ; Step 3044, bar 1397
  LIN {X 9360.893,Y -2029.899,Z 855.478,A 89.96659,B 0.00000,C 180.00000} ; outside
  LIN {X 9360.893,Y -2029.899,Z -132.531,A 89.96659,B 0.00000,C 180.00000} ; preinsert
  LIN {X 9360.893,Y -2029.899,Z -382.531,A 89.96659,B 0.00000,C 180.00000} ; insert
  LIN {X 9360.893,Y -2029.899,Z -382.531,A 89.96659,B 0.00000,C 180.00000} ; release
  LIN {X 9360.893,Y -2029.899,Z -82.531,A 89.96659,B 0.00000,C 180.00000} ; retreat
  ; Step 3045, bar 1399
  LIN {X 9485.893,Y -2029.899,Z 855.478,A 89.96659,B 0.00000,C 180.00000} ; outside
  LIN {X 9485.893,Y -2029.899,Z -132.531,A 89.96659,B 0.00000,C 180.00000} ; preinsert
  LIN {X 9485.893,Y -2029.899,Z -382.531,A 89.96659,B 0.00000,C 180.00000} ; insert
  LIN {X 9485.893,Y -2029.899,Z -382.531,A 89.96659,B 0.00000,C 180.00000} ; release
  LIN {X 9485.893,Y -2029.899,Z -82.531,A 89.96659,B 0.00000,C 180.00000} ; retreat
  ; Step 3046, bar 1401
  LIN {X 9610.893,Y -2029.899,Z 855.478,A 89.96659,B 0.00000,C 180.00000} ; outside
  LIN {X 9610.893,Y -2029.899,Z -132.531,A 89.96659,B 0.00000,C 180.00000} ; preinsert
  LIN {X 9610.893,Y -2029.899,Z -382.531,A 89.96659,B 0.00000,C 180.00000} ; insert
  LIN {X 9610.893,Y -2029.899,Z -382.531,A 89.96659,B 0.00000,C 180.00000} ; release
  LIN {X 9610.893,Y -2029.899,Z -82.531,A 89.96659,B 0.00000,C 180.00000} ; retreat
  ; Step 3047, bar 1403
  LIN {X 9735.893,Y -2029.899,Z 855.478,A 89.96659,B 0.00000,C 180.00000} ; outside
  LIN {X 9735.893,Y -2029.899,Z -132.531,A 89.96659,B 0.00000,C 180.00000} ; preinsert
  LIN {X 9735.893,Y -2029.899,Z -382.531,A 89.96659,B 0.00000,C 180.00000} ; insert
  LIN {X 9735.893,Y -2029.899,Z -382.531,A 89.96659,B 0.00000,C 180.00000} ; release
  LIN {X 9735.893,Y -2029.899,Z -82.531,A 89.96659,B 0.00000,C 180.00000} ; retreat
  ; Step 3048, bar 1405
  LIN {X 9860.893,Y -2029.899,Z 855.478,A 89.96659,B 0.00000,C 180.00000} ; outside
  LIN {X 9860.893,Y -2029.899,Z -132.531,A 89.96659,B 0.00000,C 180.00000} ; preinsert
  LIN {X 9860.893,Y -2029.899,Z -382.531,A 89.96659,B 0.00000,C 180.00000} ; insert
  LIN {X 9860.893,Y -2029.899,Z -382.531,A 89.96659,B 0.00000,C 180.00000} ; release
  LIN {X 9860.893,Y -2029.899,Z -82.531,A 89.96659,B 0.00000,C 180.00000} ; retreat
  ; Step 3049, bar 1407
  LIN {X 10110.893,Y -2029.899,Z 855.478,A 89.96659,B 0.00000,C 180.00000} ; outside
  LIN {X 10110.893,Y -2029.899,Z -132.531,A 89.96659,B 0.00000,C 180.00000} ; preinsert
  LIN {X 10110.893,Y -2029.899,Z -382.531,A 89.96659,B 0.00000,C 180.00000} ; insert
  LIN {X 10110.893,Y -2029.899,Z -382.531,A 89.96659,B 0.00000,C 180.00000} ; release
  LIN {X 10110.893,Y -2029.899,Z -82.531,A 89.96659,B 0.00000,C 180.00000} ; retreat
  ; Step 3050, bar 1409
  LIN {X 10235.893,Y -2029.899,Z 855.478,A 89.96659,B 0.00000,C 180.00000} ; outside
  LIN {X 10235.893,Y -2029.899,Z -132.531,A 89.96659,B 0.00000,C 180.00000} ; preinsert
  LIN {X 10235.893,Y -2029.899,Z -382.531,A 89.96659,B 0.00000,C 180.00000} ; insert
  LIN {X 10235.893,Y -2029.899,Z -382.531,A 89.96659,B 0.00000,C 180.00000} ; release
  LIN {X 10235.893,Y -2029.899,Z -82.531,A 89.96659,B 0.00000,C 180.00000} ; retreat
  ; Step 3051, bar 1411
  LIN {X 10360.893,Y -2029.899,Z 855.478,A 89.96659,B 0.00000,C 180.00000} ; outside
  LIN {X 10360.893,Y -2029.899,Z -132.531,A 89.96659,B 0.00000,C 180.00000} ; preinsert
  LIN {X 10360.893,Y -2029.899,Z -382.531,A 89.96659,B 0.00000,C 180.00000} ; insert
  LIN {X 10360.893,Y -2029.899,Z -382.531,A 89.96659,B 0.00000,C 180.00000} ; release
  LIN {X 10360.893,Y -2029.899,Z -82.531,A 89.96659,B 0.00000,C 180.00000} ; retreat
  ; Step 3052, bar 1413
  LIN {X 10485.893,Y -2029.899,Z 855.478,A 89.96659,B 0.00000,C 180.00000} ; outside
  LIN {X 10485.893,Y -2029.899,Z -132.531,A 89.96659,B 0.00000,C 180.00000} ; preinsert
  LIN {X 10485.893,Y -2029.899,Z -382.531,A 89.96659,B 0.00000,C 180.00000} ; insert
  LIN {X 10485.893,Y -2029.899,Z -382.531,A 89.96659,B 0.00000,C 180.00000} ; release
  LIN {X 10485.893,Y -2029.899,Z -82.531,A 89.96659,B 0.00000,C 180.00000} ; retreat
  ; Step 3053, bar 1415
  LIN {X 10610.893,Y -2029.899,Z 855.478,A 89.96659,B 0.00000,C 180.00000} ; outside
  LIN {X 10610.893,Y -2029.899,Z -132.531,A 89.96659,B 0.00000,C 180.00000} ; preinsert
  LIN {X 10610.893,Y -2029.899,Z -382.531,A 89.96659,B 0.00000,C 180.00000} ; insert
  LIN {X 10610.893,Y -2029.899,Z -382.531,A 89.96659,B 0.00000,C 180.00000} ; release
  LIN {X 10610.893,Y -2029.899,Z -82.531,A 89.96659,B 0.00000,C 180.00000} ; retreat
  ; Step 3054, bar 1417
  LIN {X 10735.893,Y -2029.899,Z 855.478,A 89.96659,B 0.00000,C 180.00000} ; outside
  LIN {X 10735.893,Y -2029.899,Z -132.531,A 89.96659,B 0.00000,C 180.00000} ; preinsert
  LIN {X 10735.893,Y -2029.899,Z -382.531,A 89.96659,B 0.00000,C 180.00000} ; insert
  LIN {X 10735.893,Y -2029.899,Z -382.531,A 89.96659,B 0.00000,C 180.00000} ; release
  LIN {X 10735.893,Y -2029.899,Z -82.531,A 89.96659,B 0.00000,C 180.00000} ; retreat
  ; Step 3055, bar 1419
  LIN {X 10860.893,Y -2029.899,Z 855.478,A 89.96659,B 0.00000,C 180.00000} ; outside
  LIN {X 10860.893,Y -2029.899,Z -132.531,A 89.96659,B 0.00000,C 180.00000} ; preinsert
  LIN {X 10860.893,Y -2029.899,Z -382.531,A 89.96659,B 0.00000,C 180.00000} ; insert
  LIN {X 10860.893,Y -2029.899,Z -382.531,A 89.96659,B 0.00000,C 180.00000} ; release
  LIN {X 10860.893,Y -2029.899,Z -82.531,A 89.96659,B 0.00000,C 180.00000} ; retreat
  ; Step 3056, bar 1421
  LIN {X 10985.893,Y -2029.899,Z 855.478,A 89.96659,B 0.00000,C 180.00000} ; outside
  LIN {X 10985.893,Y -2029.899,Z -132.531,A 89.96659,B 0.00000,C 180.00000} ; preinsert
  LIN {X 10985.893,Y -2029.899,Z -382.531,A 89.96659,B 0.00000,C 180.00000} ; insert
  LIN {X 10985.893,Y -2029.899,Z -382.531,A 89.96659,B 0.00000,C 180.00000} ; release
  LIN {X 10985.893,Y -2029.899,Z -82.531,A 89.96659,B 0.00000,C 180.00000} ; retreat
  ; Step 3057, bar 1423
  LIN {X 11110.893,Y -2029.899,Z 855.478,A 89.96659,B 0.00000,C 180.00000} ; outside
  LIN {X 11110.893,Y -2029.899,Z -132.531,A 89.96659,B 0.00000,C 180.00000} ; preinsert
  LIN {X 11110.893,Y -2029.899,Z -382.531,A 89.96659,B 0.00000,C 180.00000} ; insert
  LIN {X 11110.893,Y -2029.899,Z -382.531,A 89.96659,B 0.00000,C 180.00000} ; release
  LIN {X 11110.893,Y -2029.899,Z -82.531,A 89.96659,B 0.00000,C 180.00000} ; retreat
  ; Step 3058, bar 1425
  LIN {X 11235.893,Y -2029.899,Z 855.478,A 89.96659,B 0.00000,C 180.00000} ; outside
  LIN {X 11235.893,Y -2029.899,Z -132.531,A 89.96659,B 0.00000,C 180.00000} ; preinsert
  LIN {X 11235.893,Y -2029.899,Z -382.531,A 89.96659,B 0.00000,C 180.00000} ; insert
  LIN {X 11235.893,Y -2029.899,Z -382.531,A 89.96659,B 0.00000,C 180.00000} ; release
  LIN {X 11235.893,Y -2029.899,Z -82.531,A 89.96659,B 0.00000,C 180.00000} ; retreat
  ; Step 3059, bar 1427
  LIN {X 11360.893,Y -2029.899,Z 855.478,A 89.96659,B 0.00000,C 180.00000} ; outside
  LIN {X 11360.893,Y -2029.899,Z -132.531,A 89.96659,B 0.00000,C 180.00000} ; preinsert
  LIN {X 11360.893,Y -2029.899,Z -382.531,A 89.96659,B 0.00000,C 180.00000} ; insert
  LIN {X 11360.893,Y -2029.899,Z -382.531,A 89.96659,B 0.00000,C 180.00000} ; release
  LIN {X 11360.893,Y -2029.899,Z -82.531,A 89.96659,B 0.00000,C 180.00000} ; retreat
  ; Step 3060, bar 1429
  LIN {X 11485.893,Y -2029.899,Z 855.478,A 89.96659,B 0.00000,C 180.00000} ; outside
  LIN {X 11485.893,Y -2029.899,Z -132.531,A 89.96659,B 0.00000,C 180.00000} ; preinsert
  LIN {X 11485.893,Y -2029.899,Z -382.531,A 89.96659,B 0.00000,C 180.00000} ; insert
  LIN {X 11485.893,Y -2029.899,Z -382.531,A 89.96659,B 0.00000,C 180.00000} ; release
  LIN {X 11485.893,Y -2029.899,Z -82.531,A 89.96659,B 0.00000,C 180.00000} ; retreat
  ; Step 3061, bar 1431
  LIN {X 11610.893,Y -2029.899,Z 855.478,A 89.96659,B 0.00000,C 180.00000} ; outside
  LIN {X 11610.893,Y -2029.899,Z -132.531,A 89.96659,B 0.00000,C 180.00000} ; preinsert
  LIN {X 11610.893,Y -2029.899,Z -382.531,A 89.96659,B 0.00000,C 180.00000} ; insert
  LIN {X 11610.893,Y -2029.899,Z -382.531,A 89.96659,B 0.00000,C 180.00000} ; release
  LIN {X 11610.893,Y -2029.899,Z -82.531,A 89.96659,B 0.00000,C 180.00000} ; retreat
  ; Step 3062, bar 1433
  LIN {X 11735.893,Y -2029.899,Z 855.478,A 89.96659,B 0.00000,C 180.00000} ; outside
  LIN {X 11735.893,Y -2029.899,Z -132.531,A 89.96659,B 0.00000,C 180.00000} ; preinsert
  LIN {X 11735.893,Y -2029.899,Z -382.531,A 89.96659,B 0.00000,C 180.00000} ; insert
  LIN {X 11735.893,Y -2029.899,Z -382.531,A 89.96659,B 0.00000,C 180.00000} ; release
  LIN {X 11735.893,Y -2029.899,Z -82.531,A 89.96659,B 0.00000,C 180.00000} ; retreat
  ; Step 3063, bar 1435
  LIN {X 11860.893,Y -2029.899,Z 855.478,A 89.96659,B 0.00000,C 180.00000} ; outside
  LIN {X 11860.893,Y -2029.899,Z -132.531,A 89.96659,B 0.00000,C 180.00000} ; preinsert
  LIN {X 11860.893,Y -2029.899,Z -382.531,A 89.96659,B 0.00000,C 180.00000} ; insert
  LIN {X 11860.893,Y -2029.899,Z -382.531,A 89.96659,B 0.00000,C 180.00000} ; release
  LIN {X 11860.893,Y -2029.899,Z -82.531,A 89.96659,B 0.00000,C 180.00000} ; retreat
  ; Step 3064, bar 1437
  LIN {X 11985.893,Y -2029.899,Z 855.478,A 89.96659,B 0.00000,C 180.00000} ; outside
  LIN {X 11985.893,Y -2029.899,Z -132.531,A 89.96659,B 0.00000,C 180.00000} ; preinsert
  LIN {X 11985.893,Y -2029.899,Z -382.531,A 89.96659,B 0.00000,C 180.00000} ; insert
  LIN {X 11985.893,Y -2029.899,Z -382.531,A 89.96659,B 0.00000,C 180.00000} ; release
  LIN {X 11985.893,Y -2029.899,Z -82.531,A 89.96659,B 0.00000,C 180.00000} ; retreat
  ; Step 3065, bar 1439
  LIN {X 12110.893,Y -2029.899,Z 855.478,A 89.96659,B 0.00000,C 180.00000} ; outside
  LIN {X 12110.893,Y -2029.899,Z -132.531,A 89.96659,B 0.00000,C 180.00000} ; preinsert
  LIN {X 12110.893,Y -2029.899,Z -382.531,A 89.96659,B 0.00000,C 180.00000} ; insert
  LIN {X 12110.893,Y -2029.899,Z -382.531,A 89.96659,B 0.00000,C 180.00000} ; release
  LIN {X 12110.893,Y -2029.899,Z -82.531,A 89.96659,B 0.00000,C 180.00000} ; retreat
  ; Step 3066, bar 1441
  LIN {X 12235.893,Y -2029.899,Z 855.478,A 89.96659,B 0.00000,C 180.00000} ; outside
  LIN {X 12235.893,Y -2029.899,Z -132.531,A 89.96659,B 0.00000,C 180.00000} ; preinsert
  LIN {X 12235.893,Y -2029.899,Z -382.531,A 89.96659,B 0.00000,C 180.00000} ; insert
  LIN {X 12235.893,Y -2029.899,Z -382.531,A 89.96659,B 0.00000,C 180.00000} ; release
  LIN {X 12235.893,Y -2029.899,Z -82.531,A 89.96659,B 0.00000,C 180.00000} ; retreat
  ; Step 3067, bar 1443
  LIN {X 12335.893,Y -2029.899,Z 855.478,A 89.96659,B 0.00000,C 180.00000} ; outside
  LIN {X 12335.893,Y -2029.899,Z -132.531,A 89.96659,B 0.00000,C 180.00000} ; preinsert
  LIN {X 12335.893,Y -2029.899,Z -382.531,A 89.96659,B 0.00000,C 180.00000} ; insert
  LIN {X 12335.893,Y -2029.899,Z -382.531,A 89.96659,B 0.00000,C 180.00000} ; release
  LIN {X 12335.893,Y -2029.899,Z -82.531,A 89.96659,B 0.00000,C 180.00000} ; retreat
  ; Step 3068, bar 1445
  LIN {X 12435.893,Y -2029.899,Z 855.478,A 89.96659,B 0.00000,C 180.00000} ; outside
  LIN {X 12435.893,Y -2029.899,Z -132.531,A 89.96659,B 0.00000,C 180.00000} ; preinsert
  LIN {X 12435.893,Y -2029.899,Z -382.531,A 89.96659,B 0.00000,C 180.00000} ; insert
  LIN {X 12435.893,Y -2029.899,Z -382.531,A 89.96659,B 0.00000,C 180.00000} ; release
  LIN {X 12435.893,Y -2029.899,Z -82.531,A 89.96659,B 0.00000,C 180.00000} ; retreat
  ; Step 3069, bar 1447
  LIN {X 12535.893,Y -2029.899,Z 855.478,A 89.96659,B 0.00000,C 180.00000} ; outside
  LIN {X 12535.893,Y -2029.899,Z -132.531,A 89.96659,B 0.00000,C 180.00000} ; preinsert
  LIN {X 12535.893,Y -2029.899,Z -382.531,A 89.96659,B 0.00000,C 180.00000} ; insert
  LIN {X 12535.893,Y -2029.899,Z -382.531,A 89.96659,B 0.00000,C 180.00000} ; release
  LIN {X 12535.893,Y -2029.899,Z -82.531,A 89.96659,B 0.00000,C 180.00000} ; retreat
  ; Step 3070, bar 1449
  LIN {X 12635.893,Y -2029.899,Z 855.478,A 89.96659,B 0.00000,C 180.00000} ; outside
  LIN {X 12635.893,Y -2029.899,Z -132.531,A 89.96659,B 0.00000,C 180.00000} ; preinsert
  LIN {X 12635.893,Y -2029.899,Z -382.531,A 89.96659,B 0.00000,C 180.00000} ; insert
  LIN {X 12635.893,Y -2029.899,Z -382.531,A 89.96659,B 0.00000,C 180.00000} ; release
  LIN {X 12635.893,Y -2029.899,Z -82.531,A 89.96659,B 0.00000,C 180.00000} ; retreat
  ; Step 3071, bar 1451
  LIN {X 12735.893,Y -2029.899,Z 855.478,A 89.96659,B 0.00000,C 180.00000} ; outside
  LIN {X 12735.893,Y -2029.899,Z -132.531,A 89.96659,B 0.00000,C 180.00000} ; preinsert
  LIN {X 12735.893,Y -2029.899,Z -382.531,A 89.96659,B 0.00000,C 180.00000} ; insert
  LIN {X 12735.893,Y -2029.899,Z -382.531,A 89.96659,B 0.00000,C 180.00000} ; release
  LIN {X 12735.893,Y -2029.899,Z -82.531,A 89.96659,B 0.00000,C 180.00000} ; retreat
  ; Step 3072, bar 1453
  LIN {X 12835.893,Y -2029.899,Z 855.478,A 89.96659,B 0.00000,C 180.00000} ; outside
  LIN {X 12835.893,Y -2029.899,Z -132.531,A 89.96659,B 0.00000,C 180.00000} ; preinsert
  LIN {X 12835.893,Y -2029.899,Z -382.531,A 89.96659,B 0.00000,C 180.00000} ; insert
  LIN {X 12835.893,Y -2029.899,Z -382.531,A 89.96659,B 0.00000,C 180.00000} ; release
  LIN {X 12835.893,Y -2029.899,Z -82.531,A 89.96659,B 0.00000,C 180.00000} ; retreat
  ; Step 3073, bar 1455
  LIN {X 12935.893,Y -2029.899,Z 855.478,A 89.96659,B 0.00000,C 180.00000} ; outside
  LIN {X 12935.893,Y -2029.899,Z -132.531,A 89.96659,B 0.00000,C 180.00000} ; preinsert
  LIN {X 12935.893,Y -2029.899,Z -382.531,A 89.96659,B 0.00000,C 180.00000} ; insert
  LIN {X 12935.893,Y -2029.899,Z -382.531,A 89.96659,B 0.00000,C 180.00000} ; release
  LIN {X 12935.893,Y -2029.899,Z -82.531,A 89.96659,B 0.00000,C 180.00000} ; retreat
  ; Step 3074, bar 1457
  LIN {X 13035.893,Y -2029.899,Z 855.478,A 89.96659,B 0.00000,C 180.00000} ; outside
  LIN {X 13035.893,Y -2029.899,Z -132.531,A 89.96659,B 0.00000,C 180.00000} ; preinsert
  LIN {X 13035.893,Y -2029.899,Z -382.531,A 89.96659,B 0.00000,C 180.00000} ; insert
  LIN {X 13035.893,Y -2029.899,Z -382.531,A 89.96659,B 0.00000,C 180.00000} ; release
  LIN {X 13035.893,Y -2029.899,Z -82.531,A 89.96659,B 0.00000,C 180.00000} ; retreat
  ; Step 3075, bar 1459
  LIN {X 13135.893,Y -2029.899,Z 855.478,A 89.96659,B 0.00000,C 180.00000} ; outside
  LIN {X 13135.893,Y -2029.899,Z -132.531,A 89.96659,B 0.00000,C 180.00000} ; preinsert
  LIN {X 13135.893,Y -2029.899,Z -382.531,A 89.96659,B 0.00000,C 180.00000} ; insert
  LIN {X 13135.893,Y -2029.899,Z -382.531,A 89.96659,B 0.00000,C 180.00000} ; release
  LIN {X 13135.893,Y -2029.899,Z -82.531,A 89.96659,B 0.00000,C 180.00000} ; retreat
  ; Step 3076, bar 1461
  LIN {X 13235.893,Y -2029.899,Z 855.478,A 89.96659,B 0.00000,C 180.00000} ; outside
  LIN {X 13235.893,Y -2029.899,Z -132.531,A 89.96659,B 0.00000,C 180.00000} ; preinsert
  LIN {X 13235.893,Y -2029.899,Z -382.531,A 89.96659,B 0.00000,C 180.00000} ; insert
  LIN {X 13235.893,Y -2029.899,Z -382.531,A 89.96659,B 0.00000,C 180.00000} ; release
  LIN {X 13235.893,Y -2029.899,Z -82.531,A 89.96659,B 0.00000,C 180.00000} ; retreat
  ; Step 3077, bar 1463
  LIN {X 13335.893,Y -2029.899,Z 855.478,A 89.96659,B 0.00000,C 180.00000} ; outside
  LIN {X 13335.893,Y -2029.899,Z -132.531,A 89.96659,B 0.00000,C 180.00000} ; preinsert
  LIN {X 13335.893,Y -2029.899,Z -382.531,A 89.96659,B 0.00000,C 180.00000} ; insert
  LIN {X 13335.893,Y -2029.899,Z -382.531,A 89.96659,B 0.00000,C 180.00000} ; release
  LIN {X 13335.893,Y -2029.899,Z -82.531,A 89.96659,B 0.00000,C 180.00000} ; retreat
  ; Step 3078, bar 1465
  LIN {X 13435.893,Y -2029.899,Z 855.478,A 89.96659,B 0.00000,C 180.00000} ; outside
  LIN {X 13435.893,Y -2029.899,Z -132.531,A 89.96659,B 0.00000,C 180.00000} ; preinsert
  LIN {X 13435.893,Y -2029.899,Z -382.531,A 89.96659,B 0.00000,C 180.00000} ; insert
  LIN {X 13435.893,Y -2029.899,Z -382.531,A 89.96659,B 0.00000,C 180.00000} ; release
  LIN {X 13435.893,Y -2029.899,Z -82.531,A 89.96659,B 0.00000,C 180.00000} ; retreat
  ; Step 3079, bar 1467
  LIN {X 13535.893,Y -2029.899,Z 855.478,A 89.96659,B 0.00000,C 180.00000} ; outside
  LIN {X 13535.893,Y -2029.899,Z -132.531,A 89.96659,B 0.00000,C 180.00000} ; preinsert
  LIN {X 13535.893,Y -2029.899,Z -382.531,A 89.96659,B 0.00000,C 180.00000} ; insert
  LIN {X 13535.893,Y -2029.899,Z -382.531,A 89.96659,B 0.00000,C 180.00000} ; release
  LIN {X 13535.893,Y -2029.899,Z -82.531,A 89.96659,B 0.00000,C 180.00000} ; retreat
  ; Step 3080, bar 1469
  LIN {X 13635.893,Y -2029.899,Z 855.478,A 89.96659,B 0.00000,C 180.00000} ; outside
  LIN {X 13635.893,Y -2029.899,Z -132.531,A 89.96659,B 0.00000,C 180.00000} ; preinsert
  LIN {X 13635.893,Y -2029.899,Z -382.531,A 89.96659,B 0.00000,C 180.00000} ; insert
  LIN {X 13635.893,Y -2029.899,Z -382.531,A 89.96659,B 0.00000,C 180.00000} ; release
  LIN {X 13635.893,Y -2029.899,Z -82.531,A 89.96659,B 0.00000,C 180.00000} ; retreat
  ; Step 3081, bar 1471
  LIN {X 13735.893,Y -2029.899,Z 855.478,A 89.96659,B 0.00000,C 180.00000} ; outside
  LIN {X 13735.893,Y -2029.899,Z -132.531,A 89.96659,B 0.00000,C 180.00000} ; preinsert
  LIN {X 13735.893,Y -2029.899,Z -382.531,A 89.96659,B 0.00000,C 180.00000} ; insert
  LIN {X 13735.893,Y -2029.899,Z -382.531,A 89.96659,B 0.00000,C 180.00000} ; release
  LIN {X 13735.893,Y -2029.899,Z -82.531,A 89.96659,B 0.00000,C 180.00000} ; retreat
  ; Step 3082, bar 1473
  LIN {X 13835.893,Y -2029.899,Z 855.478,A 89.96659,B 0.00000,C 180.00000} ; outside
  LIN {X 13835.893,Y -2029.899,Z -132.531,A 89.96659,B 0.00000,C 180.00000} ; preinsert
  LIN {X 13835.893,Y -2029.899,Z -382.531,A 89.96659,B 0.00000,C 180.00000} ; insert
  LIN {X 13835.893,Y -2029.899,Z -382.531,A 89.96659,B 0.00000,C 180.00000} ; release
  LIN {X 13835.893,Y -2029.899,Z -82.531,A 89.96659,B 0.00000,C 180.00000} ; retreat
  ; Step 3083, bar 1475
  LIN {X 14135.893,Y -2029.899,Z 855.478,A 89.96659,B 0.00000,C 180.00000} ; outside
  LIN {X 14135.893,Y -2029.899,Z -132.531,A 89.96659,B 0.00000,C 180.00000} ; preinsert
  LIN {X 14135.893,Y -2029.899,Z -382.531,A 89.96659,B 0.00000,C 180.00000} ; insert
  LIN {X 14135.893,Y -2029.899,Z -382.531,A 89.96659,B 0.00000,C 180.00000} ; release
  LIN {X 14135.893,Y -2029.899,Z -82.531,A 89.96659,B 0.00000,C 180.00000} ; retreat
  ; Step 3084, bar 1477
  LIN {X 14235.893,Y -2029.899,Z 855.478,A 89.96659,B 0.00000,C 180.00000} ; outside
  LIN {X 14235.893,Y -2029.899,Z -132.531,A 89.96659,B 0.00000,C 180.00000} ; preinsert
  LIN {X 14235.893,Y -2029.899,Z -382.531,A 89.96659,B 0.00000,C 180.00000} ; insert
  LIN {X 14235.893,Y -2029.899,Z -382.531,A 89.96659,B 0.00000,C 180.00000} ; release
  LIN {X 14235.893,Y -2029.899,Z -82.531,A 89.96659,B 0.00000,C 180.00000} ; retreat
  ; Step 3085, bar 1560
  LIN {X -110.893,Y 2029.899,Z 855.478,A -90.03341,B 0.00000,C -180.00000} ; outside
  LIN {X -110.893,Y 2029.899,Z -132.531,A -90.03341,B 0.00000,C -180.00000} ; preinsert
  LIN {X -110.893,Y 2029.899,Z -382.531,A -90.03341,B 0.00000,C -180.00000} ; insert
  LIN {X -110.893,Y 2029.899,Z -382.531,A -90.03341,B 0.00000,C -180.00000} ; release
  LIN {X -110.893,Y 2029.899,Z -82.531,A -90.03341,B 0.00000,C -180.00000} ; retreat
  ; Step 3086, bar 1562
  LIN {X -235.893,Y 2029.899,Z 855.478,A -90.03341,B 0.00000,C -180.00000} ; outside
  LIN {X -235.893,Y 2029.899,Z -132.531,A -90.03341,B 0.00000,C -180.00000} ; preinsert
  LIN {X -235.893,Y 2029.899,Z -382.531,A -90.03341,B 0.00000,C -180.00000} ; insert
  LIN {X -235.893,Y 2029.899,Z -382.531,A -90.03341,B 0.00000,C -180.00000} ; release
  LIN {X -235.893,Y 2029.899,Z -82.531,A -90.03341,B 0.00000,C -180.00000} ; retreat
  ; Step 3087, bar 1564
  LIN {X -360.893,Y 2029.899,Z 855.478,A -90.03341,B 0.00000,C -180.00000} ; outside
  LIN {X -360.893,Y 2029.899,Z -132.531,A -90.03341,B 0.00000,C -180.00000} ; preinsert
  LIN {X -360.893,Y 2029.899,Z -382.531,A -90.03341,B 0.00000,C -180.00000} ; insert
  LIN {X -360.893,Y 2029.899,Z -382.531,A -90.03341,B 0.00000,C -180.00000} ; release
  LIN {X -360.893,Y 2029.899,Z -82.531,A -90.03341,B 0.00000,C -180.00000} ; retreat
  ; Step 3088, bar 1566
  LIN {X -485.893,Y 2029.899,Z 855.478,A -90.03341,B 0.00000,C -180.00000} ; outside
  LIN {X -485.893,Y 2029.899,Z -132.531,A -90.03341,B 0.00000,C -180.00000} ; preinsert
  LIN {X -485.893,Y 2029.899,Z -382.531,A -90.03341,B 0.00000,C -180.00000} ; insert
  LIN {X -485.893,Y 2029.899,Z -382.531,A -90.03341,B 0.00000,C -180.00000} ; release
  LIN {X -485.893,Y 2029.899,Z -82.531,A -90.03341,B 0.00000,C -180.00000} ; retreat
  ; Step 3089, bar 1568
  LIN {X -610.893,Y 2029.899,Z 855.478,A -90.03341,B 0.00000,C -180.00000} ; outside
  LIN {X -610.893,Y 2029.899,Z -132.531,A -90.03341,B 0.00000,C -180.00000} ; preinsert
  LIN {X -610.893,Y 2029.899,Z -382.531,A -90.03341,B 0.00000,C -180.00000} ; insert
  LIN {X -610.893,Y 2029.899,Z -382.531,A -90.03341,B 0.00000,C -180.00000} ; release
  LIN {X -610.893,Y 2029.899,Z -82.531,A -90.03341,B 0.00000,C -180.00000} ; retreat
  ; Step 3090, bar 1570
  LIN {X -735.893,Y 2029.899,Z 855.478,A -90.03341,B 0.00000,C -180.00000} ; outside
  LIN {X -735.893,Y 2029.899,Z -132.531,A -90.03341,B 0.00000,C -180.00000} ; preinsert
  LIN {X -735.893,Y 2029.899,Z -382.531,A -90.03341,B 0.00000,C -180.00000} ; insert
  LIN {X -735.893,Y 2029.899,Z -382.531,A -90.03341,B 0.00000,C -180.00000} ; release
  LIN {X -735.893,Y 2029.899,Z -82.531,A -90.03341,B 0.00000,C -180.00000} ; retreat
  ; Step 3091, bar 1572
  LIN {X -860.893,Y 2029.899,Z 855.478,A -90.03341,B 0.00000,C -180.00000} ; outside
  LIN {X -860.893,Y 2029.899,Z -132.531,A -90.03341,B 0.00000,C -180.00000} ; preinsert
  LIN {X -860.893,Y 2029.899,Z -382.531,A -90.03341,B 0.00000,C -180.00000} ; insert
  LIN {X -860.893,Y 2029.899,Z -382.531,A -90.03341,B 0.00000,C -180.00000} ; release
  LIN {X -860.893,Y 2029.899,Z -82.531,A -90.03341,B 0.00000,C -180.00000} ; retreat
  ; Step 3092, bar 1574
  LIN {X -985.893,Y 2029.899,Z 855.478,A -90.03341,B 0.00000,C -180.00000} ; outside
  LIN {X -985.893,Y 2029.899,Z -132.531,A -90.03341,B 0.00000,C -180.00000} ; preinsert
  LIN {X -985.893,Y 2029.899,Z -382.531,A -90.03341,B 0.00000,C -180.00000} ; insert
  LIN {X -985.893,Y 2029.899,Z -382.531,A -90.03341,B 0.00000,C -180.00000} ; release
  LIN {X -985.893,Y 2029.899,Z -82.531,A -90.03341,B 0.00000,C -180.00000} ; retreat
  ; Step 3093, bar 1576
  LIN {X -1110.893,Y 2029.899,Z 855.478,A -90.03341,B 0.00000,C -180.00000} ; outside
  LIN {X -1110.893,Y 2029.899,Z -132.531,A -90.03341,B 0.00000,C -180.00000} ; preinsert
  LIN {X -1110.893,Y 2029.899,Z -382.531,A -90.03341,B 0.00000,C -180.00000} ; insert
  LIN {X -1110.893,Y 2029.899,Z -382.531,A -90.03341,B 0.00000,C -180.00000} ; release
  LIN {X -1110.893,Y 2029.899,Z -82.531,A -90.03341,B 0.00000,C -180.00000} ; retreat
  ; Step 3094, bar 1578
  LIN {X -1235.893,Y 2029.899,Z 855.478,A -90.03341,B 0.00000,C -180.00000} ; outside
  LIN {X -1235.893,Y 2029.899,Z -132.531,A -90.03341,B 0.00000,C -180.00000} ; preinsert
  LIN {X -1235.893,Y 2029.899,Z -382.531,A -90.03341,B 0.00000,C -180.00000} ; insert
  LIN {X -1235.893,Y 2029.899,Z -382.531,A -90.03341,B 0.00000,C -180.00000} ; release
  LIN {X -1235.893,Y 2029.899,Z -82.531,A -90.03341,B 0.00000,C -180.00000} ; retreat
  ; Step 3095, bar 1580
  LIN {X -1360.893,Y 2029.899,Z 855.478,A -90.03341,B 0.00000,C -180.00000} ; outside
  LIN {X -1360.893,Y 2029.899,Z -132.531,A -90.03341,B 0.00000,C -180.00000} ; preinsert
  LIN {X -1360.893,Y 2029.899,Z -382.531,A -90.03341,B 0.00000,C -180.00000} ; insert
  LIN {X -1360.893,Y 2029.899,Z -382.531,A -90.03341,B 0.00000,C -180.00000} ; release
  LIN {X -1360.893,Y 2029.899,Z -82.531,A -90.03341,B 0.00000,C -180.00000} ; retreat
  ; Step 3096, bar 1582
  LIN {X -1485.893,Y 2029.899,Z 855.478,A -90.03341,B 0.00000,C -180.00000} ; outside
  LIN {X -1485.893,Y 2029.899,Z -132.531,A -90.03341,B 0.00000,C -180.00000} ; preinsert
  LIN {X -1485.893,Y 2029.899,Z -382.531,A -90.03341,B 0.00000,C -180.00000} ; insert
  LIN {X -1485.893,Y 2029.899,Z -382.531,A -90.03341,B 0.00000,C -180.00000} ; release
  LIN {X -1485.893,Y 2029.899,Z -82.531,A -90.03341,B 0.00000,C -180.00000} ; retreat
  ; Step 3097, bar 1584
  LIN {X -1610.893,Y 2029.899,Z 855.478,A -90.03341,B 0.00000,C -180.00000} ; outside
  LIN {X -1610.893,Y 2029.899,Z -132.531,A -90.03341,B 0.00000,C -180.00000} ; preinsert
  LIN {X -1610.893,Y 2029.899,Z -382.531,A -90.03341,B 0.00000,C -180.00000} ; insert
  LIN {X -1610.893,Y 2029.899,Z -382.531,A -90.03341,B 0.00000,C -180.00000} ; release
  LIN {X -1610.893,Y 2029.899,Z -82.531,A -90.03341,B 0.00000,C -180.00000} ; retreat
  ; Step 3098, bar 1586
  LIN {X -1735.893,Y 2029.899,Z 855.478,A -90.03341,B 0.00000,C -180.00000} ; outside
  LIN {X -1735.893,Y 2029.899,Z -132.531,A -90.03341,B 0.00000,C -180.00000} ; preinsert
  LIN {X -1735.893,Y 2029.899,Z -382.531,A -90.03341,B 0.00000,C -180.00000} ; insert
  LIN {X -1735.893,Y 2029.899,Z -382.531,A -90.03341,B 0.00000,C -180.00000} ; release
  LIN {X -1735.893,Y 2029.899,Z -82.531,A -90.03341,B 0.00000,C -180.00000} ; retreat
  ; Step 3099, bar 1588
  LIN {X -1860.893,Y 2029.899,Z 855.478,A -90.03341,B 0.00000,C -180.00000} ; outside
  LIN {X -1860.893,Y 2029.899,Z -132.531,A -90.03341,B 0.00000,C -180.00000} ; preinsert
  LIN {X -1860.893,Y 2029.899,Z -382.531,A -90.03341,B 0.00000,C -180.00000} ; insert
  LIN {X -1860.893,Y 2029.899,Z -382.531,A -90.03341,B 0.00000,C -180.00000} ; release
  LIN {X -1860.893,Y 2029.899,Z -82.531,A -90.03341,B 0.00000,C -180.00000} ; retreat
  ; Step 3100, bar 1590
  LIN {X -2110.893,Y 2029.899,Z 855.478,A -90.03341,B 0.00000,C -180.00000} ; outside
  LIN {X -2110.893,Y 2029.899,Z -132.531,A -90.03341,B 0.00000,C -180.00000} ; preinsert
  LIN {X -2110.893,Y 2029.899,Z -382.531,A -90.03341,B 0.00000,C -180.00000} ; insert
  LIN {X -2110.893,Y 2029.899,Z -382.531,A -90.03341,B 0.00000,C -180.00000} ; release
  LIN {X -2110.893,Y 2029.899,Z -82.531,A -90.03341,B 0.00000,C -180.00000} ; retreat
  ; Step 3101, bar 1592
  LIN {X -2235.893,Y 2029.899,Z 855.478,A -90.03341,B 0.00000,C -180.00000} ; outside
  LIN {X -2235.893,Y 2029.899,Z -132.531,A -90.03341,B 0.00000,C -180.00000} ; preinsert
  LIN {X -2235.893,Y 2029.899,Z -382.531,A -90.03341,B 0.00000,C -180.00000} ; insert
  LIN {X -2235.893,Y 2029.899,Z -382.531,A -90.03341,B 0.00000,C -180.00000} ; release
  LIN {X -2235.893,Y 2029.899,Z -82.531,A -90.03341,B 0.00000,C -180.00000} ; retreat
  ; Step 3102, bar 1594
  LIN {X -2360.893,Y 2029.899,Z 855.478,A -90.03341,B 0.00000,C -180.00000} ; outside
  LIN {X -2360.893,Y 2029.899,Z -132.531,A -90.03341,B 0.00000,C -180.00000} ; preinsert
  LIN {X -2360.893,Y 2029.899,Z -382.531,A -90.03341,B 0.00000,C -180.00000} ; insert
  LIN {X -2360.893,Y 2029.899,Z -382.531,A -90.03341,B 0.00000,C -180.00000} ; release
  LIN {X -2360.893,Y 2029.899,Z -82.531,A -90.03341,B 0.00000,C -180.00000} ; retreat
  ; Step 3103, bar 1596
  LIN {X -2485.893,Y 2029.899,Z 855.478,A -90.03341,B 0.00000,C -180.00000} ; outside
  LIN {X -2485.893,Y 2029.899,Z -132.531,A -90.03341,B 0.00000,C -180.00000} ; preinsert
  LIN {X -2485.893,Y 2029.899,Z -382.531,A -90.03341,B 0.00000,C -180.00000} ; insert
  LIN {X -2485.893,Y 2029.899,Z -382.531,A -90.03341,B 0.00000,C -180.00000} ; release
  LIN {X -2485.893,Y 2029.899,Z -82.531,A -90.03341,B 0.00000,C -180.00000} ; retreat
  ; Step 3104, bar 1598
  LIN {X -2610.893,Y 2029.899,Z 855.478,A -90.03341,B 0.00000,C -180.00000} ; outside
  LIN {X -2610.893,Y 2029.899,Z -132.531,A -90.03341,B 0.00000,C -180.00000} ; preinsert
  LIN {X -2610.893,Y 2029.899,Z -382.531,A -90.03341,B 0.00000,C -180.00000} ; insert
  LIN {X -2610.893,Y 2029.899,Z -382.531,A -90.03341,B 0.00000,C -180.00000} ; release
  LIN {X -2610.893,Y 2029.899,Z -82.531,A -90.03341,B 0.00000,C -180.00000} ; retreat
  ; Step 3105, bar 1600
  LIN {X -2735.893,Y 2029.899,Z 855.478,A -90.03341,B 0.00000,C -180.00000} ; outside
  LIN {X -2735.893,Y 2029.899,Z -132.531,A -90.03341,B 0.00000,C -180.00000} ; preinsert
  LIN {X -2735.893,Y 2029.899,Z -382.531,A -90.03341,B 0.00000,C -180.00000} ; insert
  LIN {X -2735.893,Y 2029.899,Z -382.531,A -90.03341,B 0.00000,C -180.00000} ; release
  LIN {X -2735.893,Y 2029.899,Z -82.531,A -90.03341,B 0.00000,C -180.00000} ; retreat
  ; Step 3106, bar 1602
  LIN {X -2860.893,Y 2029.899,Z 855.478,A -90.03341,B 0.00000,C -180.00000} ; outside
  LIN {X -2860.893,Y 2029.899,Z -132.531,A -90.03341,B 0.00000,C -180.00000} ; preinsert
  LIN {X -2860.893,Y 2029.899,Z -382.531,A -90.03341,B 0.00000,C -180.00000} ; insert
  LIN {X -2860.893,Y 2029.899,Z -382.531,A -90.03341,B 0.00000,C -180.00000} ; release
  LIN {X -2860.893,Y 2029.899,Z -82.531,A -90.03341,B 0.00000,C -180.00000} ; retreat
  ; Step 3107, bar 1604
  LIN {X -2985.893,Y 2029.899,Z 855.478,A -90.03341,B 0.00000,C -180.00000} ; outside
  LIN {X -2985.893,Y 2029.899,Z -132.531,A -90.03341,B 0.00000,C -180.00000} ; preinsert
  LIN {X -2985.893,Y 2029.899,Z -382.531,A -90.03341,B 0.00000,C -180.00000} ; insert
  LIN {X -2985.893,Y 2029.899,Z -382.531,A -90.03341,B 0.00000,C -180.00000} ; release
  LIN {X -2985.893,Y 2029.899,Z -82.531,A -90.03341,B 0.00000,C -180.00000} ; retreat
  ; Step 3108, bar 1606
  LIN {X -3110.893,Y 2029.899,Z 855.478,A -90.03341,B 0.00000,C -180.00000} ; outside
  LIN {X -3110.893,Y 2029.899,Z -132.531,A -90.03341,B 0.00000,C -180.00000} ; preinsert
  LIN {X -3110.893,Y 2029.899,Z -382.531,A -90.03341,B 0.00000,C -180.00000} ; insert
  LIN {X -3110.893,Y 2029.899,Z -382.531,A -90.03341,B 0.00000,C -180.00000} ; release
  LIN {X -3110.893,Y 2029.899,Z -82.531,A -90.03341,B 0.00000,C -180.00000} ; retreat
  ; Step 3109, bar 1608
  LIN {X -3235.893,Y 2029.899,Z 855.478,A -90.03341,B 0.00000,C -180.00000} ; outside
  LIN {X -3235.893,Y 2029.899,Z -132.531,A -90.03341,B 0.00000,C -180.00000} ; preinsert
  LIN {X -3235.893,Y 2029.899,Z -382.531,A -90.03341,B 0.00000,C -180.00000} ; insert
  LIN {X -3235.893,Y 2029.899,Z -382.531,A -90.03341,B 0.00000,C -180.00000} ; release
  LIN {X -3235.893,Y 2029.899,Z -82.531,A -90.03341,B 0.00000,C -180.00000} ; retreat
  ; Step 3110, bar 1610
  LIN {X -3360.893,Y 2029.899,Z 855.478,A -90.03341,B 0.00000,C -180.00000} ; outside
  LIN {X -3360.893,Y 2029.899,Z -132.531,A -90.03341,B 0.00000,C -180.00000} ; preinsert
  LIN {X -3360.893,Y 2029.899,Z -382.531,A -90.03341,B 0.00000,C -180.00000} ; insert
  LIN {X -3360.893,Y 2029.899,Z -382.531,A -90.03341,B 0.00000,C -180.00000} ; release
  LIN {X -3360.893,Y 2029.899,Z -82.531,A -90.03341,B 0.00000,C -180.00000} ; retreat
  ; Step 3111, bar 1612
  LIN {X -3485.893,Y 2029.899,Z 855.478,A -90.03341,B 0.00000,C -180.00000} ; outside
  LIN {X -3485.893,Y 2029.899,Z -132.531,A -90.03341,B 0.00000,C -180.00000} ; preinsert
  LIN {X -3485.893,Y 2029.899,Z -382.531,A -90.03341,B 0.00000,C -180.00000} ; insert
  LIN {X -3485.893,Y 2029.899,Z -382.531,A -90.03341,B 0.00000,C -180.00000} ; release
  LIN {X -3485.893,Y 2029.899,Z -82.531,A -90.03341,B 0.00000,C -180.00000} ; retreat
  ; Step 3112, bar 1614
  LIN {X -3610.893,Y 2029.899,Z 855.478,A -90.03341,B 0.00000,C -180.00000} ; outside
  LIN {X -3610.893,Y 2029.899,Z -132.531,A -90.03341,B 0.00000,C -180.00000} ; preinsert
  LIN {X -3610.893,Y 2029.899,Z -382.531,A -90.03341,B 0.00000,C -180.00000} ; insert
  LIN {X -3610.893,Y 2029.899,Z -382.531,A -90.03341,B 0.00000,C -180.00000} ; release
  LIN {X -3610.893,Y 2029.899,Z -82.531,A -90.03341,B 0.00000,C -180.00000} ; retreat
  ; Step 3113, bar 1616
  LIN {X -3735.893,Y 2029.899,Z 855.478,A -90.03341,B 0.00000,C -180.00000} ; outside
  LIN {X -3735.893,Y 2029.899,Z -132.531,A -90.03341,B 0.00000,C -180.00000} ; preinsert
  LIN {X -3735.893,Y 2029.899,Z -382.531,A -90.03341,B 0.00000,C -180.00000} ; insert
  LIN {X -3735.893,Y 2029.899,Z -382.531,A -90.03341,B 0.00000,C -180.00000} ; release
  LIN {X -3735.893,Y 2029.899,Z -82.531,A -90.03341,B 0.00000,C -180.00000} ; retreat
  ; Step 3114, bar 1618
  LIN {X -3860.893,Y 2029.899,Z 855.478,A -90.03341,B 0.00000,C -180.00000} ; outside
  LIN {X -3860.893,Y 2029.899,Z -132.531,A -90.03341,B 0.00000,C -180.00000} ; preinsert
  LIN {X -3860.893,Y 2029.899,Z -382.531,A -90.03341,B 0.00000,C -180.00000} ; insert
  LIN {X -3860.893,Y 2029.899,Z -382.531,A -90.03341,B 0.00000,C -180.00000} ; release
  LIN {X -3860.893,Y 2029.899,Z -82.531,A -90.03341,B 0.00000,C -180.00000} ; retreat
  ; Step 3115, bar 1620
  LIN {X -3985.893,Y 2029.899,Z 855.478,A -90.03341,B 0.00000,C -180.00000} ; outside
  LIN {X -3985.893,Y 2029.899,Z -132.531,A -90.03341,B 0.00000,C -180.00000} ; preinsert
  LIN {X -3985.893,Y 2029.899,Z -382.531,A -90.03341,B 0.00000,C -180.00000} ; insert
  LIN {X -3985.893,Y 2029.899,Z -382.531,A -90.03341,B 0.00000,C -180.00000} ; release
  LIN {X -3985.893,Y 2029.899,Z -82.531,A -90.03341,B 0.00000,C -180.00000} ; retreat
  ; Step 3116, bar 1622
  LIN {X -4110.893,Y 2029.899,Z 855.478,A -90.03341,B 0.00000,C -180.00000} ; outside
  LIN {X -4110.893,Y 2029.899,Z -132.531,A -90.03341,B 0.00000,C -180.00000} ; preinsert
  LIN {X -4110.893,Y 2029.899,Z -382.531,A -90.03341,B 0.00000,C -180.00000} ; insert
  LIN {X -4110.893,Y 2029.899,Z -382.531,A -90.03341,B 0.00000,C -180.00000} ; release
  LIN {X -4110.893,Y 2029.899,Z -82.531,A -90.03341,B 0.00000,C -180.00000} ; retreat
  ; Step 3117, bar 1624
  LIN {X -4235.893,Y 2029.899,Z 855.478,A -90.03341,B 0.00000,C -180.00000} ; outside
  LIN {X -4235.893,Y 2029.899,Z -132.531,A -90.03341,B 0.00000,C -180.00000} ; preinsert
  LIN {X -4235.893,Y 2029.899,Z -382.531,A -90.03341,B 0.00000,C -180.00000} ; insert
  LIN {X -4235.893,Y 2029.899,Z -382.531,A -90.03341,B 0.00000,C -180.00000} ; release
  LIN {X -4235.893,Y 2029.899,Z -82.531,A -90.03341,B 0.00000,C -180.00000} ; retreat
  ; Step 3118, bar 1626
  LIN {X -4360.893,Y 2029.899,Z 855.478,A -90.03341,B 0.00000,C -180.00000} ; outside
  LIN {X -4360.893,Y 2029.899,Z -132.531,A -90.03341,B 0.00000,C -180.00000} ; preinsert
  LIN {X -4360.893,Y 2029.899,Z -382.531,A -90.03341,B 0.00000,C -180.00000} ; insert
  LIN {X -4360.893,Y 2029.899,Z -382.531,A -90.03341,B 0.00000,C -180.00000} ; release
  LIN {X -4360.893,Y 2029.899,Z -82.531,A -90.03341,B 0.00000,C -180.00000} ; retreat
  ; Step 3119, bar 1628
  LIN {X -4485.893,Y 2029.899,Z 855.478,A -90.03341,B 0.00000,C -180.00000} ; outside
  LIN {X -4485.893,Y 2029.899,Z -132.531,A -90.03341,B 0.00000,C -180.00000} ; preinsert
  LIN {X -4485.893,Y 2029.899,Z -382.531,A -90.03341,B 0.00000,C -180.00000} ; insert
  LIN {X -4485.893,Y 2029.899,Z -382.531,A -90.03341,B 0.00000,C -180.00000} ; release
  LIN {X -4485.893,Y 2029.899,Z -82.531,A -90.03341,B 0.00000,C -180.00000} ; retreat
  ; Step 3120, bar 1630
  LIN {X -4610.893,Y 2029.899,Z 855.478,A -90.03341,B 0.00000,C -180.00000} ; outside
  LIN {X -4610.893,Y 2029.899,Z -132.531,A -90.03341,B 0.00000,C -180.00000} ; preinsert
  LIN {X -4610.893,Y 2029.899,Z -382.531,A -90.03341,B 0.00000,C -180.00000} ; insert
  LIN {X -4610.893,Y 2029.899,Z -382.531,A -90.03341,B 0.00000,C -180.00000} ; release
  LIN {X -4610.893,Y 2029.899,Z -82.531,A -90.03341,B 0.00000,C -180.00000} ; retreat
  ; Step 3121, bar 1632
  LIN {X -4735.893,Y 2029.899,Z 855.478,A -90.03341,B 0.00000,C -180.00000} ; outside
  LIN {X -4735.893,Y 2029.899,Z -132.531,A -90.03341,B 0.00000,C -180.00000} ; preinsert
  LIN {X -4735.893,Y 2029.899,Z -382.531,A -90.03341,B 0.00000,C -180.00000} ; insert
  LIN {X -4735.893,Y 2029.899,Z -382.531,A -90.03341,B 0.00000,C -180.00000} ; release
  LIN {X -4735.893,Y 2029.899,Z -82.531,A -90.03341,B 0.00000,C -180.00000} ; retreat
  ; Step 3122, bar 1634
  LIN {X -4860.893,Y 2029.899,Z 855.478,A -90.03341,B 0.00000,C -180.00000} ; outside
  LIN {X -4860.893,Y 2029.899,Z -132.531,A -90.03341,B 0.00000,C -180.00000} ; preinsert
  LIN {X -4860.893,Y 2029.899,Z -382.531,A -90.03341,B 0.00000,C -180.00000} ; insert
  LIN {X -4860.893,Y 2029.899,Z -382.531,A -90.03341,B 0.00000,C -180.00000} ; release
  LIN {X -4860.893,Y 2029.899,Z -82.531,A -90.03341,B 0.00000,C -180.00000} ; retreat
  ; Step 3123, bar 1636
  LIN {X -4985.893,Y 2029.899,Z 855.478,A -90.03341,B 0.00000,C -180.00000} ; outside
  LIN {X -4985.893,Y 2029.899,Z -132.531,A -90.03341,B 0.00000,C -180.00000} ; preinsert
  LIN {X -4985.893,Y 2029.899,Z -382.531,A -90.03341,B 0.00000,C -180.00000} ; insert
  LIN {X -4985.893,Y 2029.899,Z -382.531,A -90.03341,B 0.00000,C -180.00000} ; release
  LIN {X -4985.893,Y 2029.899,Z -82.531,A -90.03341,B 0.00000,C -180.00000} ; retreat
  ; Step 3124, bar 1638
  LIN {X -5110.893,Y 2029.899,Z 855.478,A -90.03341,B 0.00000,C -180.00000} ; outside
  LIN {X -5110.893,Y 2029.899,Z -132.531,A -90.03341,B 0.00000,C -180.00000} ; preinsert
  LIN {X -5110.893,Y 2029.899,Z -382.531,A -90.03341,B 0.00000,C -180.00000} ; insert
  LIN {X -5110.893,Y 2029.899,Z -382.531,A -90.03341,B 0.00000,C -180.00000} ; release
  LIN {X -5110.893,Y 2029.899,Z -82.531,A -90.03341,B 0.00000,C -180.00000} ; retreat
  ; Step 3125, bar 1640
  LIN {X -5235.893,Y 2029.899,Z 855.478,A -90.03341,B 0.00000,C -180.00000} ; outside
  LIN {X -5235.893,Y 2029.899,Z -132.531,A -90.03341,B 0.00000,C -180.00000} ; preinsert
  LIN {X -5235.893,Y 2029.899,Z -382.531,A -90.03341,B 0.00000,C -180.00000} ; insert
  LIN {X -5235.893,Y 2029.899,Z -382.531,A -90.03341,B 0.00000,C -180.00000} ; release
  LIN {X -5235.893,Y 2029.899,Z -82.531,A -90.03341,B 0.00000,C -180.00000} ; retreat
  ; Step 3126, bar 1642
  LIN {X -5360.893,Y 2029.899,Z 855.478,A -90.03341,B 0.00000,C -180.00000} ; outside
  LIN {X -5360.893,Y 2029.899,Z -132.531,A -90.03341,B 0.00000,C -180.00000} ; preinsert
  LIN {X -5360.893,Y 2029.899,Z -382.531,A -90.03341,B 0.00000,C -180.00000} ; insert
  LIN {X -5360.893,Y 2029.899,Z -382.531,A -90.03341,B 0.00000,C -180.00000} ; release
  LIN {X -5360.893,Y 2029.899,Z -82.531,A -90.03341,B 0.00000,C -180.00000} ; retreat
  ; Step 3127, bar 1644
  LIN {X -5485.893,Y 2029.899,Z 855.478,A -90.03341,B 0.00000,C -180.00000} ; outside
  LIN {X -5485.893,Y 2029.899,Z -132.531,A -90.03341,B 0.00000,C -180.00000} ; preinsert
  LIN {X -5485.893,Y 2029.899,Z -382.531,A -90.03341,B 0.00000,C -180.00000} ; insert
  LIN {X -5485.893,Y 2029.899,Z -382.531,A -90.03341,B 0.00000,C -180.00000} ; release
  LIN {X -5485.893,Y 2029.899,Z -82.531,A -90.03341,B 0.00000,C -180.00000} ; retreat
  ; Step 3128, bar 1646
  LIN {X -5610.893,Y 2029.899,Z 855.478,A -90.03341,B 0.00000,C -180.00000} ; outside
  LIN {X -5610.893,Y 2029.899,Z -132.531,A -90.03341,B 0.00000,C -180.00000} ; preinsert
  LIN {X -5610.893,Y 2029.899,Z -382.531,A -90.03341,B 0.00000,C -180.00000} ; insert
  LIN {X -5610.893,Y 2029.899,Z -382.531,A -90.03341,B 0.00000,C -180.00000} ; release
  LIN {X -5610.893,Y 2029.899,Z -82.531,A -90.03341,B 0.00000,C -180.00000} ; retreat
  ; Step 3129, bar 1648
  LIN {X -5735.893,Y 2029.899,Z 855.478,A -90.03341,B 0.00000,C -180.00000} ; outside
